KUKA KRL program: EPS_2_25862_MH7A_A_20251016034305.src

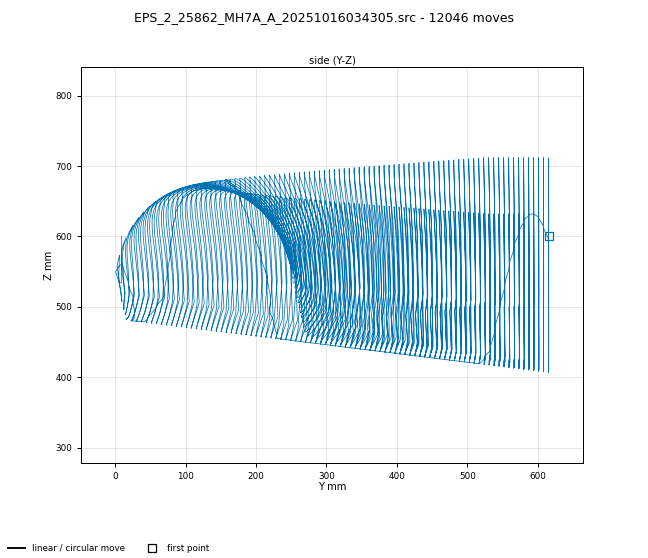
[picture p0: tool path of EPS_2_25862_MH7A_A_20251016034305.src, 12046 of 12048 moves have a stored position in this frame; points joined in program order, loops and branches not executed]
&ACCESS RVP
&REL 4
&COMMENT QRS 19112012
&PARAM EDITMASK = *
DEF PART()
EXT BAS (BAS_COMMAND :IN,REAL :IN )
INT I
BAS (#INITMOV,0 )

;KUKA QRS Post kuka4.cps  Date:22-06-2017 !

File_ID=2892

QRS_PRE_INIT()

;Init var - Until changes are made in qrs_pre_init
Outlet_Square_prg=0
Inlet_1_Square_prg=0
Inlet_2_Square_prg=0
Inlet_3_Square_prg=0
Inlet_4_Square_prg=0
Inlet_5_Square_prg=0

Outlet_1={X 0.000, Y 524.580, Z 611.500, B 0.000, E1 0.000 }
Inlet_1={X 0.000, Y 530.290, Z 531.500, B 0.000, E1 105.000 }
Outlet_1_type=201
Inlet_1_type=201
;QRS#1=Sidecore dimensions
;QRS#2=200-8" PVC SDR 35
;QRS#3=200-8" PVC SDR 35
;QRS#4=
;QRS#5=
;QRS#6=
;QRS#7=
;QRS#8=
;QRS#9=12-08 PSX
;QRS#10=12-08 PSX
;QRS#11=
;QRS#12=
;QRS#13=
;QRS#14=
;QRS#15=
;QRS#16=1220x127x991 3,25'
;QRS#17=EPS Height
;QRS#18=712
;QRS#19=*
;QRS#20= UPDATED VERSION 22-06-2017
;QRS#21=*
Outlet_Square=0100
Inlet_1_Square=0100
Inlet_2_Square=0
Inlet_3_Square=0
Inlet_4_Square=0
Inlet_5_Square=0
Mill_Square=1
Outlet_Square_Prg=204
Inlet_1_Square_prg=204

QRS_INIT()

$ADVANCE=5

; T1
PTP {E1 173.735,E2 173.735}
PTP {X 0,Y 615.512,A -85,B 0,C 180,E1 173.735,E2 173.735,E3 0,E4 0,E5 0,E6 0}
QRS_SPEED_INIT()
LIN {X 0,Y 615.512,Z 600,A -85,B 0,C 180,E1 173.735,E2 173.735,E3 0,E4 0,E5 0,E6 0} C_VEL
LIN {X 0,Y 615.512,Z 594.49,A -85,B 0,C 180,E1 173.735,E2 173.735} C_VEL
LIN {X 0,Y 615.498,Z 593.072,A -85,B 0,C 180,E1 173.417,E2 173.417} C_VEL
LIN {X 0,Y 615.497,Z 602.544,A -85,B 0,C 180,E1 172.455,E2 172.455} C_VEL
LIN {X 0,Y 615.496,Z 610.413,A -85,B 0,C 180,E1 171.464,E2 171.464} C_VEL
LIN {X 0,Y 615.497,Z 616.705,A -85,B 0,C 180,E1 170.47,E2 170.47} C_VEL
LIN {X 0,Y 615.496,Z 621.726,A -85,B 0,C 180,E1 169.473,E2 169.473} C_VEL
LIN {X 0,Y 615.496,Z 625.613,A -85,B 0,C 180,E1 168.473,E2 168.473} C_VEL
LIN {X 0,Y 615.495,Z 628.469,A -85,B 0,C 180,E1 167.47,E2 167.47} C_VEL
LIN {X 0,Y 615.496,Z 629.806,A -85,B 0,C 180,E1 166.799,E2 166.799} C_VEL
LIN {X 0,Y 615.497,Z 630.814,A -85,B 0,C 180,E1 166.065,E2 166.065} C_VEL
LIN {X 0,Y 615.494,Z 631.275,A -85,B 0,C 180,E1 165.451,E2 165.451} C_VEL
LIN {X 0,Y 615.496,Z 631.351,A -85,B 0,C 180,E1 164.774,E2 164.774} C_VEL
LIN {X 0,Y 615.495,Z 630.488,A -85,B 0,C 180,E1 163.568,E2 163.568} C_VEL
LIN {X 0,Y 615.495,Z 629.096,A -85,B 0,C 180,E1 162.73,E2 162.73} C_VEL
LIN {X 0,Y 615.497,Z 627.447,A -85,B 0,C 180,E1 162.043,E2 162.043} C_VEL
LIN {X 0,Y 615.496,Z 624.074,A -85,B 0,C 180,E1 161.009,E2 161.009} C_VEL
LIN {X 0,Y 615.496,Z 619.508,A -85,B 0,C 180,E1 159.968,E2 159.968} C_VEL
LIN {X 0,Y 615.496,Z 613.587,A -85,B 0,C 180,E1 158.919,E2 158.919} C_VEL
LIN {X 0,Y 615.498,Z 605.985,A -85,B 0,C 180,E1 157.864,E2 157.864} C_VEL
LIN {X 0,Y 615.498,Z 598.1,A -85,B 0,C 180,E1 156.978,E2 156.978} C_VEL
LIN {X 0,Y 615.497,Z 588.587,A -85,B 0,C 180,E1 156.104,E2 156.104} C_VEL
LIN {X 0,Y 615.479,Z 578.677,A -85,B 0,C 180,E1 155.368,E2 155.368} C_VEL
LIN {X 0,Y 615.462,Z 567.861,A -85,B 0,C 180,E1 154.72,E2 154.72} C_VEL
LIN {X 0,Y 615.492,Z 555.657,A -85,B 0,C 180,E1 154.148,E2 154.148} C_VEL
LIN {X 0,Y 615.484,Z 544.011,A -85,B 0,C 180,E1 153.738,E2 153.738} C_VEL
LIN {X 0,Y 615.481,Z 531.052,A -85,B 0,C 180,E1 153.424,E2 153.424} C_VEL
LIN {X 0,Y 615.492,Z 513.299,A -85,B 0,C 180,E1 153.181,E2 153.181} C_VEL
LIN {X 0,Y 615.484,Z 422.14,A -85,B 0,C 180,E1 152.108,E2 152.108} C_VEL
LIN {X 0,Y 615.478,Z 408.507,A -85,B 0,C 180,E1 149.46,E2 149.46} C_VEL
LIN {X 0,Y 615.445,Z 406.696,A -85,B 0,C 180,E1 149.078,E2 149.078} C_VEL
LIN {X 0,Y 615.439,Z 406.693,A -85,B 0,C 180,E1 146.761,E2 146.761} C_VEL
LIN {X 0,Y 615.478,Z 406.688,A -85,B 0,C 180,E1 144.168,E2 144.168} C_VEL
LIN {X 0,Y 615.489,Z 406.691,A -85,B 0,C 180,E1 141.932,E2 141.932} C_VEL
LIN {X 0,Y 615.473,Z 406.698,A -85,B 0,C 180,E1 139.392,E2 139.392} C_VEL
LIN {X 0,Y 615.443,Z 406.695,A -85,B 0,C 180,E1 136.958,E2 136.958} C_VEL
LIN {X 0,Y 615.442,Z 406.694,A -85,B 0,C 180,E1 134.927,E2 134.927} C_VEL
LIN {X 0,Y 615.485,Z 406.688,A -85,B 0,C 180,E1 132.08,E2 132.08} C_VEL
LIN {X 0,Y 615.493,Z 406.695,A -85,B 0,C 180,E1 129.75,E2 129.75} C_VEL
LIN {X 0,Y 615.444,Z 406.694,A -85,B 0,C 180,E1 126.931,E2 126.931} C_VEL
LIN {X 0,Y 615.443,Z 406.692,A -85,B 0,C 180,E1 124.694,E2 124.694} C_VEL
LIN {X 0,Y 615.46,Z 406.689,A -85,B 0,C 180,E1 122.326,E2 122.326} C_VEL
LIN {X 0,Y 615.479,Z 406.699,A -85,B 0,C 180,E1 119.407,E2 119.407} C_VEL
LIN {X 0,Y 615.447,Z 406.696,A -85,B 0,C 180,E1 117.037,E2 117.037} C_VEL
LIN {X 0,Y 615.448,Z 406.695,A -85,B 0,C 180,E1 114.994,E2 114.994} C_VEL
LIN {X 0,Y 615.462,Z 406.689,A -85,B 0,C 180,E1 112.34,E2 112.34} C_VEL
LIN {X 0,Y 615.474,Z 406.698,A -85,B 0,C 180,E1 109.339,E2 109.339} C_VEL
LIN {X 0,Y 615.468,Z 406.697,A -85,B 0,C 180,E1 107.271,E2 107.271} C_VEL
LIN {X 0,Y 615.464,Z 406.697,A -85,B 0,C 180,E1 105.227,E2 105.227} C_VEL
LIN {X 0,Y 615.462,Z 406.697,A -85,B 0,C 180,E1 103.202,E2 103.202} C_VEL
LIN {X 0,Y 615.446,Z 406.693,A -85,B 0,C 180,E1 100.867,E2 100.867} C_VEL
LIN {X 0,Y 615.45,Z 406.69,A -85,B 0,C 180,E1 98.537,E2 98.537} C_VEL
LIN {X 0,Y 615.495,Z 406.688,A -85,B 0,C 180,E1 95.899,E2 95.899} C_VEL
LIN {X 0,Y 615.471,Z 406.698,A -85,B 0,C 180,E1 93.273,E2 93.273} C_VEL
LIN {X 0,Y 615.448,Z 406.691,A -85,B 0,C 180,E1 90.655,E2 90.655} C_VEL
LIN {X 0,Y 615.495,Z 406.685,A -85,B 0,C 180,E1 88.037,E2 88.037} C_VEL
LIN {X 0,Y 615.489,Z 406.699,A -85,B 0,C 180,E1 85.416,E2 85.416} C_VEL
LIN {X 0,Y 615.446,Z 406.693,A -85,B 0,C 180,E1 82.784,E2 82.784} C_VEL
LIN {X 0,Y 615.481,Z 406.686,A -85,B 0,C 180,E1 80.138,E2 80.138} C_VEL
LIN {X 0,Y 615.487,Z 406.702,A -85,B 0,C 180,E1 77.47,E2 77.47} C_VEL
LIN {X 0,Y 615.446,Z 406.693,A -85,B 0,C 180,E1 74.773,E2 74.773} C_VEL
LIN {X 0,Y 615.49,Z 406.685,A -85,B 0,C 180,E1 72.043,E2 72.043} C_VEL
LIN {X 0,Y 615.474,Z 406.698,A -85,B 0,C 180,E1 69.269,E2 69.269} C_VEL
LIN {X 0,Y 615.466,Z 406.697,A -85,B 0,C 180,E1 67.155,E2 67.155} C_VEL
LIN {X 0,Y 615.457,Z 406.695,A -85,B 0,C 180,E1 65.007,E2 65.007} C_VEL
LIN {X 0,Y 615.451,Z 406.693,A -85,B 0,C 180,E1 62.821,E2 62.821} C_VEL
LIN {X 0,Y 615.476,Z 406.686,A -85,B 0,C 180,E1 60.208,E2 60.208} C_VEL
LIN {X 0,Y 615.493,Z 406.698,A -85,B 0,C 180,E1 57.543,E2 57.543} C_VEL
LIN {X 0,Y 615.471,Z 406.697,A -85,B 0,C 180,E1 55.184,E2 55.184} C_VEL
LIN {X 0,Y 615.451,Z 406.692,A -85,B 0,C 180,E1 52.755,E2 52.755} C_VEL
LIN {X 0,Y 615.496,Z 406.686,A -85,B 0,C 180,E1 49.91,E2 49.91} C_VEL
LIN {X 0,Y 615.493,Z 406.694,A -85,B 0,C 180,E1 47.648,E2 47.648} C_VEL
LIN {X 0,Y 615.457,Z 406.694,A -85,B 0,C 180,E1 44.929,E2 44.929} C_VEL
LIN {X 0,Y 615.487,Z 406.684,A -85,B 0,C 180,E1 42.08,E2 42.08} C_VEL
LIN {X 0,Y 615.489,Z 406.691,A -85,B 0,C 180,E1 39.75,E2 39.75} C_VEL
LIN {X 0,Y 615.458,Z 406.694,A -85,B 0,C 180,E1 36.933,E2 36.933} C_VEL
LIN {X 0,Y 615.454,Z 406.691,A -85,B 0,C 180,E1 34.696,E2 34.696} C_VEL
LIN {X 0,Y 615.465,Z 406.687,A -85,B 0,C 180,E1 32.328,E2 32.328} C_VEL
LIN {X 0,Y 615.49,Z 406.702,A -85,B 0,C 180,E1 29.406,E2 29.406} C_VEL
LIN {X 0,Y 615.464,Z 406.696,A -85,B 0,C 180,E1 27.041,E2 27.041} C_VEL
LIN {X 0,Y 615.463,Z 406.695,A -85,B 0,C 180,E1 24.993,E2 24.993} C_VEL
LIN {X 0,Y 615.466,Z 406.687,A -85,B 0,C 180,E1 22.341,E2 22.341} C_VEL
LIN {X 0,Y 615.484,Z 406.685,A -85,B 0,C 180,E1 20.033,E2 20.033} C_VEL
LIN {X 0,Y 615.487,Z 406.699,A -85,B 0,C 180,E1 17.271,E2 17.271} C_VEL
LIN {X 0,Y 615.456,Z 406.689,A -85,B 0,C 180,E1 14.55,E2 14.55} C_VEL
LIN {X 0,Y 615.494,Z 406.686,A -85,B 0,C 180,E1 11.861,E2 11.861} C_VEL
LIN {X 0,Y 615.482,Z 406.698,A -85,B 0,C 180,E1 9.199,E2 9.199} C_VEL
LIN {X 0,Y 615.458,Z 406.689,A -85,B 0,C 180,E1 6.555,E2 6.555} C_VEL
LIN {X 0,Y 615.489,Z 406.685,A -85,B 0,C 180,E1 3.928,E2 3.928} C_VEL
LIN {X 0,Y 615.494,Z 406.7,A -85,B 0,C 180,E1 1.309,E2 1.309} C_VEL
LIN {X 0,Y 615.458,Z 406.691,A -85,B 0,C 180,E1 -1.309,E2 -1.309} C_VEL
LIN {X 0,Y 615.485,Z 406.684,A -85,B 0,C 180,E1 -3.929,E2 -3.929} C_VEL
LIN {X 0,Y 615.489,Z 406.699,A -85,B 0,C 180,E1 -6.579,E2 -6.579} C_VEL
LIN {X 0,Y 615.46,Z 406.693,A -85,B 0,C 180,E1 -9.199,E2 -9.199} C_VEL
LIN {X 0,Y 615.485,Z 406.683,A -85,B 0,C 180,E1 -11.861,E2 -11.861} C_VEL
LIN {X 0,Y 615.489,Z 406.698,A -85,B 0,C 180,E1 -14.549,E2 -14.549} C_VEL
LIN {X 0,Y 615.458,Z 406.692,A -85,B 0,C 180,E1 -17.271,E2 -17.271} C_VEL
LIN {X 0,Y 615.489,Z 406.684,A -85,B 0,C 180,E1 -20.033,E2 -20.033} C_VEL
LIN {X 0,Y 615.484,Z 406.698,A -85,B 0,C 180,E1 -22.845,E2 -22.845} C_VEL
LIN {X 0,Y 615.465,Z 406.687,A -85,B 0,C 180,E1 -25.565,E2 -25.565} C_VEL
LIN {X 0,Y 615.484,Z 406.694,A -85,B 0,C 180,E1 -28.45,E2 -28.45} C_VEL
LIN {X 0,Y 615.468,Z 406.694,A -85,B 0,C 180,E1 -31.083,E2 -31.083} C_VEL
LIN {X 0,Y 615.464,Z 406.688,A -85,B 0,C 180,E1 -33.531,E2 -33.531} C_VEL
LIN {X 0,Y 615.483,Z 406.683,A -85,B 0,C 180,E1 -35.833,E2 -35.833} C_VEL
LIN {X 0,Y 615.487,Z 406.684,A -85,B 0,C 180,E1 -38.069,E2 -38.069} C_VEL
LIN {X 0,Y 615.485,Z 406.699,A -85,B 0,C 180,E1 -40.607,E2 -40.607} C_VEL
LIN {X 0,Y 615.464,Z 406.692,A -85,B 0,C 180,E1 -43.247,E2 -43.247} C_VEL
LIN {X 0,Y 615.487,Z 406.683,A -85,B 0,C 180,E1 -46.003,E2 -46.003} C_VEL
LIN {X 0,Y 615.48,Z 406.698,A -85,B 0,C 180,E1 -48.907,E2 -48.907} C_VEL
LIN {X 0,Y 615.471,Z 406.695,A -85,B 0,C 180,E1 -51.095,E2 -51.095} C_VEL
LIN {X 0,Y 615.467,Z 406.687,A -85,B 0,C 180,E1 -53.574,E2 -53.574} C_VEL
LIN {X 0,Y 615.487,Z 406.692,A -85,B 0,C 180,E1 -56.466,E2 -56.466} C_VEL
LIN {X 0,Y 615.47,Z 406.696,A -85,B 0,C 180,E1 -59.079,E2 -59.079} C_VEL
LIN {X 0,Y 615.467,Z 406.687,A -85,B 0,C 180,E1 -61.554,E2 -61.554} C_VEL
LIN {X 0,Y 615.486,Z 406.691,A -85,B 0,C 180,E1 -64.432,E2 -64.432} C_VEL
LIN {X 0,Y 615.49,Z 406.748,A -85,B 0,C 180,E1 -66.02,E2 -66.02} C_VEL
LIN {X 0,Y 615.457,Z 428.81,A -85,B 0,C 180,E1 -68.743,E2 -68.743} C_VEL
LIN {X 0,Y 615.492,Z 450.661,A -85,B 0,C 180,E1 -71.395,E2 -71.395} C_VEL
LIN {X 0,Y 615.489,Z 474.676,A -85,B 0,C 180,E1 -74.265,E2 -74.265} C_VEL
LIN {X 0,Y 615.443,Z 497.572,A -85,B 0,C 180,E1 -76.966,E2 -76.966} C_VEL
LIN {X 0,Y 615.447,Z 498.822,A -85,B 0,C 180,E1 -77.113,E2 -77.113} C_VEL
LIN {X 0,Y 615.467,Z 607.846,A -85,B 0,C 180,E1 -78.41,E2 -78.41} C_VEL
LIN {X 0,Y 615.463,Z 620.356,A -85,B 0,C 180,E1 -78.682,E2 -78.682} C_VEL
LIN {X 0,Y 615.484,Z 633.665,A -85,B 0,C 180,E1 -79.115,E2 -79.115} C_VEL
LIN {X 0,Y 615.486,Z 645.481,A -85,B 0,C 180,E1 -79.64,E2 -79.64} C_VEL
LIN {X 0,Y 615.492,Z 656.998,A -85,B 0,C 180,E1 -80.304,E2 -80.304} C_VEL
LIN {X 0,Y 615.499,Z 667.344,A -85,B 0,C 180,E1 -81.05,E2 -81.05} C_VEL
LIN {X 0,Y 615.498,Z 675.814,A -85,B 0,C 180,E1 -81.794,E2 -81.794} C_VEL
LIN {X 0,Y 615.498,Z 683.608,A -85,B 0,C 180,E1 -82.62,E2 -82.62} C_VEL
LIN {X 0,Y 615.496,Z 691.204,A -85,B 0,C 180,E1 -83.608,E2 -83.608} C_VEL
LIN {X 0,Y 615.498,Z 698.206,A -85,B 0,C 180,E1 -84.759,E2 -84.759} C_VEL
LIN {X 0,Y 615.494,Z 702.852,A -85,B 0,C 180,E1 -85.744,E2 -85.744} C_VEL
LIN {X 0,Y 615.494,Z 706.399,A -85,B 0,C 180,E1 -86.727,E2 -86.727} C_VEL
LIN {X 0,Y 615.497,Z 708.233,A -85,B 0,C 180,E1 -87.382,E2 -87.382} C_VEL
LIN {X 0,Y 615.499,Z 709.608,A -85,B 0,C 180,E1 -88.037,E2 -88.037} C_VEL
LIN {X 0,Y 615.496,Z 711.174,A -85,B 0,C 180,E1 -89.346,E2 -89.346} C_VEL
LIN {X 0,Y 615.494,Z 711.389,A -85,B 0,C 180,E1 -90,E2 -90} C_VEL
LIN {X 0,Y 615.495,Z 710.58,A -85,B 0,C 180,E1 -91.309,E2 -91.309} C_VEL
LIN {X 0,Y 615.499,Z 709.607,A -85,B 0,C 180,E1 -91.963,E2 -91.963} C_VEL
LIN {X 0,Y 615.497,Z 708.232,A -85,B 0,C 180,E1 -92.618,E2 -92.618} C_VEL
LIN {X 0,Y 615.496,Z 705.349,A -85,B 0,C 180,E1 -93.601,E2 -93.601} C_VEL
LIN {X 0,Y 615.498,Z 701.44,A -85,B 0,C 180,E1 -94.585,E2 -94.585} C_VEL
LIN {X 0,Y 615.499,Z 696.403,A -85,B 0,C 180,E1 -95.57,E2 -95.57} C_VEL
LIN {X 0,Y 615.497,Z 689.87,A -85,B 0,C 180,E1 -96.583,E2 -96.583} C_VEL
LIN {X 0,Y 615.497,Z 682.131,A -85,B 0,C 180,E1 -97.546,E2 -97.546} C_VEL
LIN {X 0,Y 615.498,Z 674.042,A -85,B 0,C 180,E1 -98.371,E2 -98.371} C_VEL
LIN {X 0,Y 615.499,Z 664.164,A -85,B 0,C 180,E1 -99.199,E2 -99.199} C_VEL
LIN {X 0,Y 615.491,Z 652.976,A -85,B 0,C 180,E1 -99.945,E2 -99.945} C_VEL
LIN {X 0,Y 615.487,Z 642.017,A -85,B 0,C 180,E1 -100.527,E2 -100.527} C_VEL
LIN {X 0,Y 615.473,Z 629.513,A -85,B 0,C 180,E1 -101.04,E2 -101.04} C_VEL
LIN {X 0,Y 615.463,Z 617.058,A -85,B 0,C 180,E1 -101.402,E2 -101.402} C_VEL
LIN {X 0,Y 615.47,Z 603.45,A -85,B 0,C 180,E1 -101.653,E2 -101.653} C_VEL
LIN {X 0,Y 615.447,Z 498.818,A -85,B 0,C 180,E1 -102.888,E2 -102.888} C_VEL
LIN {X 0,Y 615.492,Z 476.104,A -85,B 0,C 180,E1 -105.566,E2 -105.566} C_VEL
LIN {X 0,Y 615.494,Z 452.01,A -85,B 0,C 180,E1 -108.443,E2 -108.443} C_VEL
LIN {X 0,Y 615.447,Z 430.241,A -85,B 0,C 180,E1 -111.083,E2 -111.083} C_VEL
LIN {X 0,Y 615.487,Z 408.335,A -85,B 0,C 180,E1 -113.783,E2 -113.783} C_VEL
LIN {X 0,Y 615.492,Z 406.682,A -85,B 0,C 180,E1 -114.009,E2 -114.009} C_VEL
LIN {X 0,Y 615.471,Z 406.688,A -85,B 0,C 180,E1 -116.445,E2 -116.445} C_VEL
LIN {X 0,Y 615.471,Z 406.693,A -85,B 0,C 180,E1 -118.659,E2 -118.659} C_VEL
LIN {X 0,Y 615.484,Z 406.702,A -85,B 0,C 180,E1 -121.085,E2 -121.085} C_VEL
LIN {X 0,Y 615.493,Z 406.681,A -85,B 0,C 180,E1 -124.022,E2 -124.022} C_VEL
LIN {X 0,Y 615.485,Z 406.703,A -85,B 0,C 180,E1 -126.936,E2 -126.936} C_VEL
LIN {X 0,Y 615.476,Z 406.686,A -85,B 0,C 180,E1 -129.751,E2 -129.751} C_VEL
LIN {X 0,Y 615.485,Z 406.69,A -85,B 0,C 180,E1 -132.354,E2 -132.354} C_VEL
LIN {X 0,Y 615.471,Z 406.695,A -85,B 0,C 180,E1 -135.071,E2 -135.071} C_VEL
LIN {X 0,Y 615.488,Z 406.684,A -85,B 0,C 180,E1 -137.92,E2 -137.92} C_VEL
LIN {X 0,Y 615.491,Z 406.69,A -85,B 0,C 180,E1 -140.25,E2 -140.25} C_VEL
LIN {X 0,Y 615.456,Z 406.695,A -85,B 0,C 180,E1 -143.068,E2 -143.068} C_VEL
LIN {X 0,Y 615.449,Z 406.692,A -85,B 0,C 180,E1 -145.305,E2 -145.305} C_VEL
LIN {X 0,Y 615.461,Z 406.69,A -85,B 0,C 180,E1 -147.674,E2 -147.674} C_VEL
LIN {X 0,Y 615.473,Z 406.699,A -85,B 0,C 180,E1 -150.593,E2 -150.593} C_VEL
LIN {X 0,Y 615.44,Z 406.696,A -85,B 0,C 180,E1 -152.965,E2 -152.965} C_VEL
LIN {X 0,Y 615.432,Z 406.697,A -85,B 0,C 180,E1 -155.006,E2 -155.006} C_VEL
LIN {X 0,Y 615.429,Z 406.696,A -85,B 0,C 180,E1 -157.153,E2 -157.153} C_VEL
LIN {X 0,Y 615.483,Z 406.697,A -85,B 0,C 180,E1 -159.967,E2 -159.967} C_VEL
LIN {X 0,Y 615.428,Z 406.699,A -85,B 0,C 180,E1 -162.728,E2 -162.728} C_VEL
LIN {X 0,Y 615.42,Z 406.7,A -85,B 0,C 180,E1 -164.772,E2 -164.772} C_VEL
LIN {X 0,Y 615.415,Z 406.7,A -85,B 0,C 180,E1 -166.797,E2 -166.797} C_VEL
LIN {X 0,Y 615.416,Z 406.7,A -85,B 0,C 180,E1 -169.149,E2 -169.149} C_VEL
LIN {X 0,Y 615.442,Z 406.699,A -85,B 0,C 180,E1 -171.463,E2 -171.463} C_VEL
LIN {X 0,Y 615.483,Z 406.695,A -85,B 0,C 180,E1 -174.101,E2 -174.101} C_VEL
LIN {X 0,Y 615.43,Z 406.696,A -85,B 0,C 180,E1 -176.727,E2 -176.727} C_VEL
LIN {X 0,Y 615.442,Z 406.697,A -85,B 0,C 180,E1 -179.182,E2 -179.182} C_VEL
LIN {X 0,Y 615.474,Z 419.232,A -85,B 0,C 180,E1 -181.636,E2 -181.636} C_VEL
LIN {X 0,Y 615.482,Z 422.09,A -85,B 0,C 180,E1 -182.188,E2 -182.188} C_VEL
LIN {X 0,Y 615.485,Z 527.922,A -85,B 0,C 180,E1 -183.457,E2 -183.457} C_VEL
LIN {X 0,Y 615.482,Z 540.23,A -85,B 0,C 180,E1 -183.724,E2 -183.724} C_VEL
LIN {X 0,Y 615.496,Z 552.949,A -85,B 0,C 180,E1 -184.133,E2 -184.133} C_VEL
LIN {X 0,Y 615.468,Z 565.139,A -85,B 0,C 180,E1 -184.667,E2 -184.667} C_VEL
LIN {X 0,Y 615.471,Z 576.613,A -85,B 0,C 180,E1 -185.323,E2 -185.323} C_VEL
LIN {X 0,Y 615.498,Z 586.934,A -85,B 0,C 180,E1 -186.063,E2 -186.063} C_VEL
LIN {X 0,Y 615.498,Z 593.072,A -85,B 0,C 180,E1 -186.583,E2 -186.583} C_VEL
LIN {X 0,Y 614.841,Z 597.363,A -85,B 0,C 180,E1 -186.973,E2 -186.973} C_VEL
LIN {X 0,Y 611.975,Z 603.961,A -85,B 0,C 180,E1 -187.622,E2 -187.622} C_VEL
LIN {X 0,Y 609.116,Z 609.736,A -85,B 0,C 180,E1 -188.318,E2 -188.318} C_VEL
LIN {X 0,Y 608.449,Z 612.931,A -85,B 0,C 180,E1 -188.774,E2 -188.774} C_VEL
LIN {X 0,Y 608.433,Z 618.129,A -85,B 0,C 180,E1 -189.642,E2 -189.642} C_VEL
LIN {X 0,Y 608.437,Z 622.99,A -85,B 0,C 180,E1 -190.65,E2 -190.65} C_VEL
LIN {X 0,Y 608.436,Z 626.725,A -85,B 0,C 180,E1 -191.662,E2 -191.662} C_VEL
LIN {X 0,Y 608.419,Z 629.431,A -85,B 0,C 180,E1 -192.678,E2 -192.678} C_VEL
LIN {X 0,Y 608.439,Z 630.696,A -85,B 0,C 180,E1 -193.357,E2 -193.357} C_VEL
LIN {X 0,Y 608.435,Z 631.54,A -85,B 0,C 180,E1 -194.038,E2 -194.038} C_VEL
LIN {X 0,Y 608.424,Z 631.93,A -85,B 0,C 180,E1 -194.722,E2 -194.722} C_VEL
LIN {X 0,Y 608.419,Z 631.921,A -85,B 0,C 180,E1 -195.407,E2 -195.407} C_VEL
LIN {X 0,Y 608.422,Z 631.014,A -85,B 0,C 180,E1 -196.513,E2 -196.513} C_VEL
LIN {X 0,Y 608.42,Z 629.289,A -85,B 0,C 180,E1 -197.478,E2 -197.478} C_VEL
LIN {X 0,Y 608.429,Z 625.843,A -85,B 0,C 180,E1 -198.703,E2 -198.703} C_VEL
LIN {X 0,Y 608.435,Z 620.813,A -85,B 0,C 180,E1 -199.923,E2 -199.923} C_VEL
LIN {X 0,Y 608.452,Z 615.05,A -85,B 0,C 180,E1 -200.982,E2 -200.982} C_VEL
LIN {X 0,Y 608.456,Z 607.715,A -85,B 0,C 180,E1 -202.049,E2 -202.049} C_VEL
LIN {X 0,Y 608.457,Z 600.081,A -85,B 0,C 180,E1 -202.944,E2 -202.944} C_VEL
LIN {X 0,Y 608.482,Z 590.643,A -85,B 0,C 180,E1 -203.844,E2 -203.844} C_VEL
LIN {X 0,Y 608.479,Z 580.109,A -85,B 0,C 180,E1 -204.661,E2 -204.661} C_VEL
LIN {X 0,Y 608.468,Z 568.498,A -85,B 0,C 180,E1 -205.373,E2 -205.373} C_VEL
LIN {X 0,Y 608.508,Z 556.778,A -85,B 0,C 180,E1 -205.935,E2 -205.935} C_VEL
LIN {X 0,Y 608.526,Z 543.817,A -85,B 0,C 180,E1 -206.401,E2 -206.401} C_VEL
LIN {X 0,Y 608.537,Z 530.376,A -85,B 0,C 180,E1 -206.724,E2 -206.724} C_VEL
LIN {X 0,Y 608.556,Z 509.869,A -85,B 0,C 180,E1 -206.997,E2 -206.997} C_VEL
LIN {X 0,Y 608.446,Z 422.357,A -85,B 0,C 180,E1 -208.044,E2 -208.044} C_VEL
LIN {X 0,Y 608.451,Z 408.589,A -85,B 0,C 180,E1 -210.738,E2 -210.738} C_VEL
LIN {X 0,Y 608.416,Z 407.694,A -85,B 0,C 180,E1 -210.933,E2 -210.933} C_VEL
LIN {X 0,Y 608.437,Z 407.692,A -85,B 0,C 180,E1 -212.881,E2 -212.881} C_VEL
LIN {X 0,Y 608.416,Z 407.692,A -85,B 0,C 180,E1 -215.28,E2 -215.28} C_VEL
LIN {X 0,Y 608.465,Z 407.694,A -85,B 0,C 180,E1 -218.239,E2 -218.239} C_VEL
LIN {X 0,Y 608.412,Z 407.693,A -85,B 0,C 180,E1 -221.18,E2 -221.18} C_VEL
LIN {X 0,Y 608.465,Z 407.688,A -85,B 0,C 180,E1 -223.87,E2 -223.87} C_VEL
LIN {X 0,Y 608.452,Z 407.693,A -85,B 0,C 180,E1 -226.693,E2 -226.693} C_VEL
LIN {X 0,Y 608.426,Z 407.694,A -85,B 0,C 180,E1 -228.821,E2 -228.821} C_VEL
LIN {X 0,Y 608.457,Z 407.688,A -85,B 0,C 180,E1 -231.761,E2 -231.761} C_VEL
LIN {X 0,Y 608.434,Z 407.695,A -85,B 0,C 180,E1 -234.721,E2 -234.721} C_VEL
LIN {X 0,Y 608.434,Z 407.69,A -85,B 0,C 180,E1 -237.119,E2 -237.119} C_VEL
LIN {X 0,Y 608.471,Z 407.689,A -85,B 0,C 180,E1 -240.028,E2 -240.028} C_VEL
LIN {X 0,Y 608.454,Z 407.691,A -85,B 0,C 180,E1 -242.798,E2 -242.798} C_VEL
LIN {X 0,Y 608.431,Z 407.69,A -85,B 0,C 180,E1 -245.428,E2 -245.428} C_VEL
LIN {X 0,Y 608.467,Z 407.694,A -85,B 0,C 180,E1 -248.308,E2 -248.308} C_VEL
LIN {X 0,Y 608.438,Z 407.69,A -85,B 0,C 180,E1 -251.13,E2 -251.13} C_VEL
LIN {X 0,Y 608.455,Z 407.689,A -85,B 0,C 180,E1 -253.906,E2 -253.906} C_VEL
LIN {X 0,Y 608.449,Z 407.695,A -85,B 0,C 180,E1 -256.643,E2 -256.643} C_VEL
LIN {X 0,Y 608.43,Z 407.69,A -85,B 0,C 180,E1 -259.349,E2 -259.349} C_VEL
LIN {X 0,Y 608.48,Z 407.687,A -85,B 0,C 180,E1 -262.033,E2 -262.033} C_VEL
LIN {X 0,Y 608.451,Z 407.694,A -85,B 0,C 180,E1 -264.698,E2 -264.698} C_VEL
LIN {X 0,Y 608.444,Z 407.688,A -85,B 0,C 180,E1 -267.352,E2 -267.352} C_VEL
LIN {X 0,Y 608.477,Z 407.687,A -85,B 0,C 180,E1 -270,E2 -270} C_VEL
LIN {X 0,Y 608.474,Z 407.693,A -85,B 0,C 180,E1 -272.648,E2 -272.648} C_VEL
LIN {X 0,Y 608.433,Z 407.69,A -85,B 0,C 180,E1 -275.302,E2 -275.302} C_VEL
LIN {X 0,Y 608.475,Z 407.687,A -85,B 0,C 180,E1 -277.967,E2 -277.967} C_VEL
LIN {X 0,Y 608.429,Z 407.694,A -85,B 0,C 180,E1 -280.935,E2 -280.935} C_VEL
LIN {X 0,Y 608.437,Z 407.689,A -85,B 0,C 180,E1 -283.357,E2 -283.357} C_VEL
LIN {X 0,Y 608.46,Z 407.69,A -85,B 0,C 180,E1 -286.094,E2 -286.094} C_VEL
LIN {X 0,Y 608.448,Z 407.692,A -85,B 0,C 180,E1 -288.87,E2 -288.87} C_VEL
LIN {X 0,Y 608.453,Z 407.687,A -85,B 0,C 180,E1 -291.692,E2 -291.692} C_VEL
LIN {X 0,Y 608.446,Z 407.698,A -85,B 0,C 180,E1 -294.571,E2 -294.571} C_VEL
LIN {X 0,Y 608.431,Z 407.691,A -85,B 0,C 180,E1 -297.198,E2 -297.198} C_VEL
LIN {X 0,Y 608.461,Z 407.686,A -85,B 0,C 180,E1 -299.78,E2 -299.78} C_VEL
LIN {X 0,Y 608.466,Z 407.696,A -85,B 0,C 180,E1 -302.523,E2 -302.523} C_VEL
LIN {X 0,Y 608.425,Z 407.691,A -85,B 0,C 180,E1 -305.279,E2 -305.279} C_VEL
LIN {X 0,Y 608.466,Z 407.691,A -85,B 0,C 180,E1 -308.24,E2 -308.24} C_VEL
LIN {X 0,Y 608.424,Z 407.692,A -85,B 0,C 180,E1 -311.179,E2 -311.179} C_VEL
LIN {X 0,Y 608.466,Z 407.686,A -85,B 0,C 180,E1 -313.87,E2 -313.87} C_VEL
LIN {X 0,Y 608.468,Z 407.694,A -85,B 0,C 180,E1 -316.691,E2 -316.691} C_VEL
LIN {X 0,Y 608.44,Z 407.695,A -85,B 0,C 180,E1 -318.822,E2 -318.822} C_VEL
LIN {X 0,Y 608.46,Z 407.686,A -85,B 0,C 180,E1 -321.76,E2 -321.76} C_VEL
LIN {X 0,Y 608.447,Z 407.689,A -85,B 0,C 180,E1 -323.954,E2 -323.954} C_VEL
LIN {X 0,Y 608.47,Z 407.691,A -85,B 0,C 180,E1 -326.33,E2 -326.33} C_VEL
LIN {X 0,Y 608.443,Z 407.697,A -85,B 0,C 180,E1 -328.733,E2 -328.733} C_VEL
LIN {X 0,Y 608.449,Z 407.688,A -85,B 0,C 180,E1 -331.384,E2 -331.384} C_VEL
LIN {X 0,Y 608.437,Z 407.69,A -85,B 0,C 180,E1 -333.964,E2 -333.964} C_VEL
LIN {X 0,Y 608.473,Z 407.688,A -85,B 0,C 180,E1 -336.155,E2 -336.155} C_VEL
LIN {X 0,Y 608.444,Z 407.692,A -85,B 0,C 180,E1 -339.018,E2 -339.018} C_VEL
LIN {X 0,Y 608.444,Z 407.689,A -85,B 0,C 180,E1 -341.828,E2 -341.828} C_VEL
LIN {X 0,Y 608.467,Z 407.696,A -85,B 0,C 180,E1 -344.594,E2 -344.594} C_VEL
LIN {X 0,Y 608.454,Z 407.688,A -85,B 0,C 180,E1 -347.323,E2 -347.323} C_VEL
LIN {X 0,Y 608.456,Z 407.688,A -85,B 0,C 180,E1 -350.023,E2 -350.023} C_VEL
LIN {X 0,Y 608.462,Z 407.696,A -85,B 0,C 180,E1 -352.701,E2 -352.701} C_VEL
LIN {X 0,Y 608.467,Z 407.695,A -85,B 0,C 180,E1 -354.698,E2 -354.698} C_VEL
LIN {X 0,Y 608.452,Z 407.688,A -85,B 0,C 180,E1 -357.352,E2 -357.352} C_VEL
LIN {X 0,Y 608.477,Z 407.685,A -85,B 0,C 180,E1 -360,E2 -360} C_VEL
LIN {X 0,Y 608.48,Z 407.695,A -85,B 0,C 180,E1 -362.648,E2 -362.648} C_VEL
LIN {X 0,Y 608.443,Z 407.69,A -85,B 0,C 180,E1 -365.302,E2 -365.302} C_VEL
LIN {X 0,Y 608.477,Z 407.685,A -85,B 0,C 180,E1 -367.967,E2 -367.967} C_VEL
LIN {X 0,Y 608.465,Z 407.691,A -85,B 0,C 180,E1 -370.954,E2 -370.954} C_VEL
LIN {X 0,Y 608.446,Z 407.689,A -85,B 0,C 180,E1 -373.357,E2 -373.357} C_VEL
LIN {X 0,Y 608.461,Z 407.688,A -85,B 0,C 180,E1 -376.094,E2 -376.094} C_VEL
LIN {X 0,Y 608.452,Z 407.695,A -85,B 0,C 180,E1 -378.87,E2 -378.87} C_VEL
LIN {X 0,Y 608.457,Z 407.686,A -85,B 0,C 180,E1 -381.692,E2 -381.692} C_VEL
LIN {X 0,Y 608.449,Z 407.696,A -85,B 0,C 180,E1 -384.571,E2 -384.571} C_VEL
LIN {X 0,Y 608.442,Z 407.691,A -85,B 0,C 180,E1 -387.201,E2 -387.201} C_VEL
LIN {X 0,Y 608.465,Z 407.686,A -85,B 0,C 180,E1 -389.971,E2 -389.971} C_VEL
LIN {X 0,Y 608.448,Z 407.696,A -85,B 0,C 180,E1 -392.88,E2 -392.88} C_VEL
LIN {X 0,Y 608.435,Z 407.691,A -85,B 0,C 180,E1 -395.278,E2 -395.278} C_VEL
LIN {X 0,Y 608.468,Z 407.688,A -85,B 0,C 180,E1 -398.24,E2 -398.24} C_VEL
LIN {X 0,Y 608.437,Z 407.692,A -85,B 0,C 180,E1 -401.178,E2 -401.178} C_VEL
LIN {X 0,Y 608.467,Z 407.685,A -85,B 0,C 180,E1 -403.87,E2 -403.87} C_VEL
LIN {X 0,Y 608.483,Z 407.694,A -85,B 0,C 180,E1 -406.69,E2 -406.69} C_VEL
LIN {X 0,Y 608.451,Z 407.697,A -85,B 0,C 180,E1 -408.823,E2 -408.823} C_VEL
LIN {X 0,Y 608.431,Z 407.691,A -85,B 0,C 180,E1 -411.409,E2 -411.409} C_VEL
LIN {X 0,Y 608.448,Z 407.688,A -85,B 0,C 180,E1 -413.955,E2 -413.955} C_VEL
LIN {X 0,Y 608.466,Z 407.689,A -85,B 0,C 180,E1 -416.33,E2 -416.33} C_VEL
LIN {X 0,Y 608.448,Z 407.698,A -85,B 0,C 180,E1 -418.733,E2 -418.733} C_VEL
LIN {X 0,Y 608.456,Z 407.688,A -85,B 0,C 180,E1 -421.383,E2 -421.383} C_VEL
LIN {X 0,Y 608.438,Z 407.69,A -85,B 0,C 180,E1 -423.964,E2 -423.964} C_VEL
LIN {X 0,Y 608.48,Z 407.711,A -85,B 0,C 180,E1 -425.848,E2 -425.848} C_VEL
LIN {X 0,Y 608.595,Z 424.505,A -85,B 0,C 180,E1 -427.957,E2 -427.957} C_VEL
LIN {X 0,Y 608.525,Z 447.466,A -85,B 0,C 180,E1 -430.783,E2 -430.783} C_VEL
LIN {X 0,Y 608.505,Z 468.571,A -85,B 0,C 180,E1 -433.34,E2 -433.34} C_VEL
LIN {X 0,Y 608.503,Z 491.694,A -85,B 0,C 180,E1 -436.103,E2 -436.103} C_VEL
LIN {X 0,Y 608.478,Z 499.265,A -85,B 0,C 180,E1 -436.973,E2 -436.973} C_VEL
LIN {X 0,Y 608.531,Z 607.958,A -85,B 0,C 180,E1 -438.277,E2 -438.277} C_VEL
LIN {X 0,Y 608.498,Z 621.224,A -85,B 0,C 180,E1 -438.571,E2 -438.571} C_VEL
LIN {X 0,Y 608.512,Z 633.649,A -85,B 0,C 180,E1 -438.983,E2 -438.983} C_VEL
LIN {X 0,Y 608.504,Z 645.639,A -85,B 0,C 180,E1 -439.519,E2 -439.519} C_VEL
LIN {X 0,Y 608.483,Z 657.2,A -85,B 0,C 180,E1 -440.191,E2 -440.191} C_VEL
LIN {X 0,Y 608.485,Z 667.596,A -85,B 0,C 180,E1 -440.946,E2 -440.946} C_VEL
LIN {X 0,Y 608.475,Z 676.114,A -85,B 0,C 180,E1 -441.699,E2 -441.699} C_VEL
LIN {X 0,Y 608.471,Z 683.962,A -85,B 0,C 180,E1 -442.534,E2 -442.534} C_VEL
LIN {X 0,Y 608.461,Z 691.287,A -85,B 0,C 180,E1 -443.485,E2 -443.485} C_VEL
LIN {X 0,Y 608.45,Z 696.867,A -85,B 0,C 180,E1 -444.366,E2 -444.366} C_VEL
LIN {X 0,Y 608.432,Z 701.951,A -85,B 0,C 180,E1 -445.362,E2 -445.362} C_VEL
LIN {X 0,Y 608.449,Z 705.897,A -85,B 0,C 180,E1 -446.358,E2 -446.358} C_VEL
LIN {X 0,Y 608.425,Z 708.81,A -85,B 0,C 180,E1 -447.352,E2 -447.352} C_VEL
LIN {X 0,Y 608.444,Z 710.202,A -85,B 0,C 180,E1 -448.014,E2 -448.014} C_VEL
LIN {X 0,Y 608.438,Z 711.784,A -85,B 0,C 180,E1 -449.338,E2 -449.338} C_VEL
LIN {X 0,Y 608.434,Z 712,A -85,B 0,C 180,E1 -450,E2 -450} C_VEL
LIN {X 0,Y 608.448,Z 711.183,A -85,B 0,C 180,E1 -451.324,E2 -451.324} C_VEL
LIN {X 0,Y 608.444,Z 710.201,A -85,B 0,C 180,E1 -451.986,E2 -451.986} C_VEL
LIN {X 0,Y 608.425,Z 708.808,A -85,B 0,C 180,E1 -452.649,E2 -452.649} C_VEL
LIN {X 0,Y 608.449,Z 705.895,A -85,B 0,C 180,E1 -453.643,E2 -453.643} C_VEL
LIN {X 0,Y 608.432,Z 701.949,A -85,B 0,C 180,E1 -454.638,E2 -454.638} C_VEL
LIN {X 0,Y 608.437,Z 695.875,A -85,B 0,C 180,E1 -455.801,E2 -455.801} C_VEL
LIN {X 0,Y 608.462,Z 689.233,A -85,B 0,C 180,E1 -456.8,E2 -456.8} C_VEL
LIN {X 0,Y 608.456,Z 680.987,A -85,B 0,C 180,E1 -457.8,E2 -457.8} C_VEL
LIN {X 0,Y 608.472,Z 672.533,A -85,B 0,C 180,E1 -458.636,E2 -458.636} C_VEL
LIN {X 0,Y 608.478,Z 662.087,A -85,B 0,C 180,E1 -459.474,E2 -459.474} C_VEL
LIN {X 0,Y 608.501,Z 651.751,A -85,B 0,C 180,E1 -460.145,E2 -460.145} C_VEL
LIN {X 0,Y 608.517,Z 640.598,A -85,B 0,C 180,E1 -460.725,E2 -460.725} C_VEL
LIN {X 0,Y 608.515,Z 628.894,A -85,B 0,C 180,E1 -461.192,E2 -461.192} C_VEL
LIN {X 0,Y 608.528,Z 616.254,A -85,B 0,C 180,E1 -461.555,E2 -461.555} C_VEL
LIN {X 0,Y 608.533,Z 603.581,A -85,B 0,C 180,E1 -461.787,E2 -461.787} C_VEL
LIN {X 0,Y 608.446,Z 498.943,A -85,B 0,C 180,E1 -463.038,E2 -463.038} C_VEL
LIN {X 0,Y 608.503,Z 476.162,A -85,B 0,C 180,E1 -465.749,E2 -465.749} C_VEL
LIN {X 0,Y 608.558,Z 453.372,A -85,B 0,C 180,E1 -468.497,E2 -468.497} C_VEL
LIN {X 0,Y 608.537,Z 431.676,A -85,B 0,C 180,E1 -471.156,E2 -471.156} C_VEL
LIN {X 0,Y 608.622,Z 410.151,A -85,B 0,C 180,E1 -473.839,E2 -473.839} C_VEL
LIN {X 0,Y 608.47,Z 407.688,A -85,B 0,C 180,E1 -474.168,E2 -474.168} C_VEL
LIN {X 0,Y 608.446,Z 407.693,A -85,B 0,C 180,E1 -476.775,E2 -476.775} C_VEL
LIN {X 0,Y 608.471,Z 407.686,A -85,B 0,C 180,E1 -479.78,E2 -479.78} C_VEL
LIN {X 0,Y 608.454,Z 407.69,A -85,B 0,C 180,E1 -482.521,E2 -482.521} C_VEL
LIN {X 0,Y 608.453,Z 407.698,A -85,B 0,C 180,E1 -484.906,E2 -484.906} C_VEL
LIN {X 0,Y 608.467,Z 407.686,A -85,B 0,C 180,E1 -487.747,E2 -487.747} C_VEL
LIN {X 0,Y 608.455,Z 407.69,A -85,B 0,C 180,E1 -490.329,E2 -490.329} C_VEL
LIN {X 0,Y 608.445,Z 407.696,A -85,B 0,C 180,E1 -492.961,E2 -492.961} C_VEL
LIN {X 0,Y 608.454,Z 407.687,A -85,B 0,C 180,E1 -495.737,E2 -495.737} C_VEL
LIN {X 0,Y 608.459,Z 407.697,A -85,B 0,C 180,E1 -498.659,E2 -498.659} C_VEL
LIN {X 0,Y 608.461,Z 407.687,A -85,B 0,C 180,E1 -501.761,E2 -501.761} C_VEL
LIN {X 0,Y 608.436,Z 407.696,A -85,B 0,C 180,E1 -504.722,E2 -504.722} C_VEL
LIN {X 0,Y 608.438,Z 407.691,A -85,B 0,C 180,E1 -507.119,E2 -507.119} C_VEL
LIN {X 0,Y 608.471,Z 407.69,A -85,B 0,C 180,E1 -510.029,E2 -510.029} C_VEL
LIN {X 0,Y 608.426,Z 407.694,A -85,B 0,C 180,E1 -512.803,E2 -512.803} C_VEL
LIN {X 0,Y 608.42,Z 407.695,A -85,B 0,C 180,E1 -514.697,E2 -514.697} C_VEL
LIN {X 0,Y 608.416,Z 407.693,A -85,B 0,C 180,E1 -516.875,E2 -516.875} C_VEL
LIN {X 0,Y 608.428,Z 407.691,A -85,B 0,C 180,E1 -519.332,E2 -519.332} C_VEL
LIN {X 0,Y 608.436,Z 407.695,A -85,B 0,C 180,E1 -521.828,E2 -521.828} C_VEL
LIN {X 0,Y 608.426,Z 407.693,A -85,B 0,C 180,E1 -524.593,E2 -524.593} C_VEL
LIN {X 0,Y 608.412,Z 407.694,A -85,B 0,C 180,E1 -526.642,E2 -526.642} C_VEL
LIN {X 0,Y 608.385,Z 407.696,A -85,B 0,C 180,E1 -529.087,E2 -529.087} C_VEL
LIN {X 0,Y 608.414,Z 407.695,A -85,B 0,C 180,E1 -531.363,E2 -531.363} C_VEL
LIN {X 0,Y 608.453,Z 407.695,A -85,B 0,C 180,E1 -534.033,E2 -534.033} C_VEL
LIN {X 0,Y 608.403,Z 407.694,A -85,B 0,C 180,E1 -536.689,E2 -536.689} C_VEL
LIN {X 0,Y 608.422,Z 407.694,A -85,B 0,C 180,E1 -539.173,E2 -539.173} C_VEL
LIN {X 0,Y 608.443,Z 420.348,A -85,B 0,C 180,E1 -541.655,E2 -541.655} C_VEL
LIN {X 0,Y 608.446,Z 422.367,A -85,B 0,C 180,E1 -542.048,E2 -542.048} C_VEL
LIN {X 0,Y 608.533,Z 528.482,A -85,B 0,C 180,E1 -543.331,E2 -543.331} C_VEL
LIN {X 0,Y 608.542,Z 541.347,A -85,B 0,C 180,E1 -543.621,E2 -543.621} C_VEL
LIN {X 0,Y 608.537,Z 554.388,A -85,B 0,C 180,E1 -544.056,E2 -544.056} C_VEL
LIN {X 0,Y 608.474,Z 565.459,A -85,B 0,C 180,E1 -544.554,E2 -544.554} C_VEL
LIN {X 0,Y 608.457,Z 576.937,A -85,B 0,C 180,E1 -545.219,E2 -545.219} C_VEL
LIN {X 0,Y 608.498,Z 587.278,A -85,B 0,C 180,E1 -545.967,E2 -545.967} C_VEL
LIN {X 0,Y 608.463,Z 596.693,A -85,B 0,C 180,E1 -546.799,E2 -546.799} C_VEL
LIN {X 0,Y 608.455,Z 605.778,A -85,B 0,C 180,E1 -547.8,E2 -547.8} C_VEL
LIN {X 0,Y 608.449,Z 612.931,A -85,B 0,C 180,E1 -548.774,E2 -548.774} C_VEL
LIN {X 0,Y 607.782,Z 615.966,A -85,B 0,C 180,E1 -549.248,E2 -549.248} C_VEL
LIN {X 0,Y 604.898,Z 620.355,A -85,B 0,C 180,E1 -550.044,E2 -550.044} C_VEL
LIN {X 0,Y 602.005,Z 624.121,A -85,B 0,C 180,E1 -550.877,E2 -550.877} C_VEL
LIN {X 0,Y 601.332,Z 626.018,A -85,B 0,C 180,E1 -551.406,E2 -551.406} C_VEL
LIN {X 0,Y 601.338,Z 628.229,A -85,B 0,C 180,E1 -552.144,E2 -552.144} C_VEL
LIN {X 0,Y 601.325,Z 629.813,A -85,B 0,C 180,E1 -552.83,E2 -552.83} C_VEL
LIN {X 0,Y 601.353,Z 631.568,A -85,B 0,C 180,E1 -554.064,E2 -554.064} C_VEL
LIN {X 0,Y 601.319,Z 631.972,A -85,B 0,C 180,E1 -554.9,E2 -554.9} C_VEL
LIN {X 0,Y 601.326,Z 631.858,A -85,B 0,C 180,E1 -555.594,E2 -555.594} C_VEL
LIN {X 0,Y 601.322,Z 630.94,A -85,B 0,C 180,E1 -556.587,E2 -556.587} C_VEL
LIN {X 0,Y 601.314,Z 628.884,A -85,B 0,C 180,E1 -557.691,E2 -557.691} C_VEL
LIN {X 0,Y 601.348,Z 625.663,A -85,B 0,C 180,E1 -558.798,E2 -558.798} C_VEL
LIN {X 0,Y 601.336,Z 621.621,A -85,B 0,C 180,E1 -559.812,E2 -559.812} C_VEL
LIN {X 0,Y 601.382,Z 615.68,A -85,B 0,C 180,E1 -560.947,E2 -560.947} C_VEL
LIN {X 0,Y 601.377,Z 608.969,A -85,B 0,C 180,E1 -561.961,E2 -561.961} C_VEL
LIN {X 0,Y 601.405,Z 601.62,A -85,B 0,C 180,E1 -562.865,E2 -562.865} C_VEL
LIN {X 0,Y 601.446,Z 592.622,A -85,B 0,C 180,E1 -563.775,E2 -563.775} C_VEL
LIN {X 0,Y 601.458,Z 582.107,A -85,B 0,C 180,E1 -564.629,E2 -564.629} C_VEL
LIN {X 0,Y 601.446,Z 571.279,A -85,B 0,C 180,E1 -565.339,E2 -565.339} C_VEL
LIN {X 0,Y 601.544,Z 559.517,A -85,B 0,C 180,E1 -565.944,E2 -565.944} C_VEL
LIN {X 0,Y 601.569,Z 546.444,A -85,B 0,C 180,E1 -566.449,E2 -566.449} C_VEL
LIN {X 0,Y 601.591,Z 533.518,A -85,B 0,C 180,E1 -566.799,E2 -566.799} C_VEL
LIN {X 0,Y 601.614,Z 520.564,A -85,B 0,C 180,E1 -567.009,E2 -567.009} C_VEL
LIN {X 0,Y 601.529,Z 423.337,A -85,B 0,C 180,E1 -568.176,E2 -568.176} C_VEL
LIN {X 0,Y 601.388,Z 422.349,A -85,B 0,C 180,E1 -568.201,E2 -568.201} C_VEL
LIN {X 0,Y 601.393,Z 408.996,A -85,B 0,C 180,E1 -570.846,E2 -570.846} C_VEL
LIN {X 0,Y 601.389,Z 408.57,A -85,B 0,C 180,E1 -570.944,E2 -570.944} C_VEL
LIN {X 0,Y 601.41,Z 408.564,A -85,B 0,C 180,E1 -573.315,E2 -573.315} C_VEL
LIN {X 0,Y 601.394,Z 408.575,A -85,B 0,C 180,E1 -576.259,E2 -576.259} C_VEL
LIN {X 0,Y 601.384,Z 408.568,A -85,B 0,C 180,E1 -579.129,E2 -579.129} C_VEL
LIN {X 0,Y 601.419,Z 408.565,A -85,B 0,C 180,E1 -581.766,E2 -581.766} C_VEL
LIN {X 0,Y 601.401,Z 408.574,A -85,B 0,C 180,E1 -584.532,E2 -584.532} C_VEL
LIN {X 0,Y 601.372,Z 408.569,A -85,B 0,C 180,E1 -587.414,E2 -587.414} C_VEL
LIN {X 0,Y 601.402,Z 408.569,A -85,B 0,C 180,E1 -590.004,E2 -590.004} C_VEL
LIN {X 0,Y 601.402,Z 408.573,A -85,B 0,C 180,E1 -592.622,E2 -592.622} C_VEL
LIN {X 0,Y 601.381,Z 408.569,A -85,B 0,C 180,E1 -595.065,E2 -595.065} C_VEL
LIN {X 0,Y 601.405,Z 408.565,A -85,B 0,C 180,E1 -597.482,E2 -597.482} C_VEL
LIN {X 0,Y 601.409,Z 408.566,A -85,B 0,C 180,E1 -599.855,E2 -599.855} C_VEL
LIN {X 0,Y 601.399,Z 408.573,A -85,B 0,C 180,E1 -602.641,E2 -602.641} C_VEL
LIN {X 0,Y 601.387,Z 408.568,A -85,B 0,C 180,E1 -605.12,E2 -605.12} C_VEL
LIN {X 0,Y 601.399,Z 408.57,A -85,B 0,C 180,E1 -608.04,E2 -608.04} C_VEL
LIN {X 0,Y 601.409,Z 408.568,A -85,B 0,C 180,E1 -610.9,E2 -610.9} C_VEL
LIN {X 0,Y 601.414,Z 408.565,A -85,B 0,C 180,E1 -613.712,E2 -613.712} C_VEL
LIN {X 0,Y 601.409,Z 408.575,A -85,B 0,C 180,E1 -616.484,E2 -616.484} C_VEL
LIN {X 0,Y 601.388,Z 408.568,A -85,B 0,C 180,E1 -619.223,E2 -619.223} C_VEL
LIN {X 0,Y 601.439,Z 408.563,A -85,B 0,C 180,E1 -621.939,E2 -621.939} C_VEL
LIN {X 0,Y 601.417,Z 408.571,A -85,B 0,C 180,E1 -624.636,E2 -624.636} C_VEL
LIN {X 0,Y 601.413,Z 408.564,A -85,B 0,C 180,E1 -627.321,E2 -627.321} C_VEL
LIN {X 0,Y 601.445,Z 408.563,A -85,B 0,C 180,E1 -630,E2 -630} C_VEL
LIN {X 0,Y 601.437,Z 408.568,A -85,B 0,C 180,E1 -632.679,E2 -632.679} C_VEL
LIN {X 0,Y 601.401,Z 408.566,A -85,B 0,C 180,E1 -635.364,E2 -635.364} C_VEL
LIN {X 0,Y 601.438,Z 408.564,A -85,B 0,C 180,E1 -638.061,E2 -638.061} C_VEL
LIN {X 0,Y 601.405,Z 408.568,A -85,B 0,C 180,E1 -641.001,E2 -641.001} C_VEL
LIN {X 0,Y 601.4,Z 408.566,A -85,B 0,C 180,E1 -643.516,E2 -643.516} C_VEL
LIN {X 0,Y 601.441,Z 408.567,A -85,B 0,C 180,E1 -646.287,E2 -646.287} C_VEL
LIN {X 0,Y 601.41,Z 408.566,A -85,B 0,C 180,E1 -649.099,E2 -649.099} C_VEL
LIN {X 0,Y 601.395,Z 408.567,A -85,B 0,C 180,E1 -651.24,E2 -651.24} C_VEL
LIN {X 0,Y 601.463,Z 408.562,A -85,B 0,C 180,E1 -654.14,E2 -654.14} C_VEL
LIN {X 0,Y 601.393,Z 408.568,A -85,B 0,C 180,E1 -657.114,E2 -657.114} C_VEL
LIN {X 0,Y 601.396,Z 408.566,A -85,B 0,C 180,E1 -659.394,E2 -659.394} C_VEL
LIN {X 0,Y 601.398,Z 408.566,A -85,B 0,C 180,E1 -661.727,E2 -661.727} C_VEL
LIN {X 0,Y 601.42,Z 408.567,A -85,B 0,C 180,E1 -664.119,E2 -664.119} C_VEL
LIN {X 0,Y 601.392,Z 408.577,A -85,B 0,C 180,E1 -666.584,E2 -666.584} C_VEL
LIN {X 0,Y 601.396,Z 408.568,A -85,B 0,C 180,E1 -669.128,E2 -669.128} C_VEL
LIN {X 0,Y 601.42,Z 408.563,A -85,B 0,C 180,E1 -671.765,E2 -671.765} C_VEL
LIN {X 0,Y 601.425,Z 408.573,A -85,B 0,C 180,E1 -674.535,E2 -674.535} C_VEL
LIN {X 0,Y 601.38,Z 408.569,A -85,B 0,C 180,E1 -677.327,E2 -677.327} C_VEL
LIN {X 0,Y 601.401,Z 408.567,A -85,B 0,C 180,E1 -680.004,E2 -680.004} C_VEL
LIN {X 0,Y 601.432,Z 408.572,A -85,B 0,C 180,E1 -682.618,E2 -682.618} C_VEL
LIN {X 0,Y 601.39,Z 408.57,A -85,B 0,C 180,E1 -685.066,E2 -685.066} C_VEL
LIN {X 0,Y 601.41,Z 408.564,A -85,B 0,C 180,E1 -687.483,E2 -687.483} C_VEL
LIN {X 0,Y 601.429,Z 408.563,A -85,B 0,C 180,E1 -689.851,E2 -689.851} C_VEL
LIN {X 0,Y 601.42,Z 408.569,A -85,B 0,C 180,E1 -692.887,E2 -692.887} C_VEL
LIN {X 0,Y 601.457,Z 408.559,A -85,B 0,C 180,E1 -695.86,E2 -695.86} C_VEL
LIN {X 0,Y 601.403,Z 408.573,A -85,B 0,C 180,E1 -698.761,E2 -698.761} C_VEL
LIN {X 0,Y 601.411,Z 408.564,A -85,B 0,C 180,E1 -701.608,E2 -701.608} C_VEL
LIN {X 0,Y 601.41,Z 408.571,A -85,B 0,C 180,E1 -704.409,E2 -704.409} C_VEL
LIN {X 0,Y 601.404,Z 408.567,A -85,B 0,C 180,E1 -707.171,E2 -707.171} C_VEL
LIN {X 0,Y 601.429,Z 408.563,A -85,B 0,C 180,E1 -709.905,E2 -709.905} C_VEL
LIN {X 0,Y 601.44,Z 408.571,A -85,B 0,C 180,E1 -712.615,E2 -712.615} C_VEL
LIN {X 0,Y 601.401,Z 408.567,A -85,B 0,C 180,E1 -715.308,E2 -715.308} C_VEL
LIN {X 0,Y 601.434,Z 408.563,A -85,B 0,C 180,E1 -717.991,E2 -717.991} C_VEL
LIN {X 0,Y 601.452,Z 408.57,A -85,B 0,C 180,E1 -720.67,E2 -720.67} C_VEL
LIN {X 0,Y 601.408,Z 408.566,A -85,B 0,C 180,E1 -723.35,E2 -723.35} C_VEL
LIN {X 0,Y 601.415,Z 408.565,A -85,B 0,C 180,E1 -726.037,E2 -726.037} C_VEL
LIN {X 0,Y 601.415,Z 408.574,A -85,B 0,C 180,E1 -728.738,E2 -728.738} C_VEL
LIN {X 0,Y 601.409,Z 408.565,A -85,B 0,C 180,E1 -731.459,E2 -731.459} C_VEL
LIN {X 0,Y 601.42,Z 408.566,A -85,B 0,C 180,E1 -734.206,E2 -734.206} C_VEL
LIN {X 0,Y 601.428,Z 408.568,A -85,B 0,C 180,E1 -736.986,E2 -736.986} C_VEL
LIN {X 0,Y 601.399,Z 408.566,A -85,B 0,C 180,E1 -739.81,E2 -739.81} C_VEL
LIN {X 0,Y 601.416,Z 408.573,A -85,B 0,C 180,E1 -742.606,E2 -742.606} C_VEL
LIN {X 0,Y 601.394,Z 408.574,A -85,B 0,C 180,E1 -744.879,E2 -744.879} C_VEL
LIN {X 0,Y 601.393,Z 408.568,A -85,B 0,C 180,E1 -747.358,E2 -747.358} C_VEL
LIN {X 0,Y 601.413,Z 408.565,A -85,B 0,C 180,E1 -749.394,E2 -749.394} C_VEL
LIN {X 0,Y 601.399,Z 408.566,A -85,B 0,C 180,E1 -751.727,E2 -751.727} C_VEL
LIN {X 0,Y 601.423,Z 408.565,A -85,B 0,C 180,E1 -754.119,E2 -754.119} C_VEL
LIN {X 0,Y 601.403,Z 408.574,A -85,B 0,C 180,E1 -756.583,E2 -756.583} C_VEL
LIN {X 0,Y 601.404,Z 408.569,A -85,B 0,C 180,E1 -759.127,E2 -759.127} C_VEL
LIN {X 0,Y 601.422,Z 408.563,A -85,B 0,C 180,E1 -761.766,E2 -761.766} C_VEL
LIN {X 0,Y 601.426,Z 408.57,A -85,B 0,C 180,E1 -764.535,E2 -764.535} C_VEL
LIN {X 0,Y 601.406,Z 408.567,A -85,B 0,C 180,E1 -767.329,E2 -767.329} C_VEL
LIN {X 0,Y 601.412,Z 408.565,A -85,B 0,C 180,E1 -770.005,E2 -770.005} C_VEL
LIN {X 0,Y 601.436,Z 408.57,A -85,B 0,C 180,E1 -772.618,E2 -772.618} C_VEL
LIN {X 0,Y 601.399,Z 408.571,A -85,B 0,C 180,E1 -775.067,E2 -775.067} C_VEL
LIN {X 0,Y 601.416,Z 408.564,A -85,B 0,C 180,E1 -777.484,E2 -777.484} C_VEL
LIN {X 0,Y 601.43,Z 408.562,A -85,B 0,C 180,E1 -779.852,E2 -779.852} C_VEL
LIN {X 0,Y 601.449,Z 408.569,A -85,B 0,C 180,E1 -782.889,E2 -782.889} C_VEL
LIN {X 0,Y 601.44,Z 408.581,A -85,B 0,C 180,E1 -785.658,E2 -785.658} C_VEL
LIN {X 0,Y 601.76,Z 411.59,A -85,B 0,C 180,E1 -786.056,E2 -786.056} C_VEL
LIN {X 0,Y 601.649,Z 431.68,A -85,B 0,C 180,E1 -788.59,E2 -788.59} C_VEL
LIN {X 0,Y 601.609,Z 453.123,A -85,B 0,C 180,E1 -791.251,E2 -791.251} C_VEL
LIN {X 0,Y 601.532,Z 477.601,A -85,B 0,C 180,E1 -794.238,E2 -794.238} C_VEL
LIN {X 0,Y 601.436,Z 498.947,A -85,B 0,C 180,E1 -796.807,E2 -796.807} C_VEL
LIN {X 0,Y 601.634,Z 525.202,A -85,B 0,C 180,E1 -797.134,E2 -797.134} C_VEL
LIN {X 0,Y 601.602,Z 607.958,A -85,B 0,C 180,E1 -798.14,E2 -798.14} C_VEL
LIN {X 0,Y 601.562,Z 621.224,A -85,B 0,C 180,E1 -798.438,E2 -798.438} C_VEL
LIN {X 0,Y 601.543,Z 632.916,A -85,B 0,C 180,E1 -798.826,E2 -798.826} C_VEL
LIN {X 0,Y 601.516,Z 645.638,A -85,B 0,C 180,E1 -799.396,E2 -799.396} C_VEL
LIN {X 0,Y 601.484,Z 657.202,A -85,B 0,C 180,E1 -800.076,E2 -800.076} C_VEL
LIN {X 0,Y 601.444,Z 667.598,A -85,B 0,C 180,E1 -800.839,E2 -800.839} C_VEL
LIN {X 0,Y 601.429,Z 676.114,A -85,B 0,C 180,E1 -801.601,E2 -801.601} C_VEL
LIN {X 0,Y 601.418,Z 683.962,A -85,B 0,C 180,E1 -802.446,E2 -802.446} C_VEL
LIN {X 0,Y 601.37,Z 691.226,A -85,B 0,C 180,E1 -803.398,E2 -803.398} C_VEL
LIN {X 0,Y 601.372,Z 696.867,A -85,B 0,C 180,E1 -804.299,E2 -804.299} C_VEL
LIN {X 0,Y 601.336,Z 701.951,A -85,B 0,C 180,E1 -805.308,E2 -805.308} C_VEL
LIN {X 0,Y 601.368,Z 705.897,A -85,B 0,C 180,E1 -806.315,E2 -806.315} C_VEL
LIN {X 0,Y 601.325,Z 708.81,A -85,B 0,C 180,E1 -807.321,E2 -807.321} C_VEL
LIN {X 0,Y 601.343,Z 710.202,A -85,B 0,C 180,E1 -807.991,E2 -807.991} C_VEL
LIN {X 0,Y 601.339,Z 711.784,A -85,B 0,C 180,E1 -809.331,E2 -809.331} C_VEL
LIN {X 0,Y 601.335,Z 712,A -85,B 0,C 180,E1 -810,E2 -810} C_VEL
LIN {X 0,Y 601.347,Z 711.184,A -85,B 0,C 180,E1 -811.34,E2 -811.34} C_VEL
LIN {X 0,Y 601.343,Z 710.201,A -85,B 0,C 180,E1 -812.01,E2 -812.01} C_VEL
LIN {X 0,Y 601.325,Z 708.809,A -85,B 0,C 180,E1 -812.68,E2 -812.68} C_VEL
LIN {X 0,Y 601.368,Z 705.895,A -85,B 0,C 180,E1 -813.686,E2 -813.686} C_VEL
LIN {X 0,Y 601.336,Z 701.949,A -85,B 0,C 180,E1 -814.693,E2 -814.693} C_VEL
LIN {X 0,Y 601.372,Z 695.875,A -85,B 0,C 180,E1 -815.869,E2 -815.869} C_VEL
LIN {X 0,Y 601.382,Z 689.233,A -85,B 0,C 180,E1 -816.88,E2 -816.88} C_VEL
LIN {X 0,Y 601.401,Z 680.987,A -85,B 0,C 180,E1 -817.893,E2 -817.893} C_VEL
LIN {X 0,Y 601.436,Z 672.534,A -85,B 0,C 180,E1 -818.738,E2 -818.738} C_VEL
LIN {X 0,Y 601.448,Z 662.088,A -85,B 0,C 180,E1 -819.585,E2 -819.585} C_VEL
LIN {X 0,Y 601.478,Z 651.752,A -85,B 0,C 180,E1 -820.265,E2 -820.265} C_VEL
LIN {X 0,Y 601.535,Z 640.908,A -85,B 0,C 180,E1 -820.835,E2 -820.835} C_VEL
LIN {X 0,Y 601.545,Z 628.375,A -85,B 0,C 180,E1 -821.341,E2 -821.341} C_VEL
LIN {X 0,Y 601.554,Z 615.34,A -85,B 0,C 180,E1 -821.712,E2 -821.712} C_VEL
LIN {X 0,Y 601.61,Z 602.062,A -85,B 0,C 180,E1 -821.946,E2 -821.946} C_VEL
LIN {X 0,Y 601.466,Z 499.224,A -85,B 0,C 180,E1 -823.182,E2 -823.182} C_VEL
LIN {X 0,Y 601.532,Z 477.597,A -85,B 0,C 180,E1 -825.762,E2 -825.762} C_VEL
LIN {X 0,Y 601.61,Z 453.121,A -85,B 0,C 180,E1 -828.749,E2 -828.749} C_VEL
LIN {X 0,Y 601.65,Z 431.676,A -85,B 0,C 180,E1 -831.41,E2 -831.41} C_VEL
LIN {X 0,Y 601.76,Z 411.586,A -85,B 0,C 180,E1 -833.945,E2 -833.945} C_VEL
LIN {X 0,Y 601.422,Z 408.568,A -85,B 0,C 180,E1 -834.362,E2 -834.362} C_VEL
LIN {X 0,Y 601.454,Z 408.57,A -85,B 0,C 180,E1 -837.111,E2 -837.111} C_VEL
LIN {X 0,Y 601.432,Z 408.563,A -85,B 0,C 180,E1 -840.164,E2 -840.164} C_VEL
LIN {X 0,Y 601.417,Z 408.57,A -85,B 0,C 180,E1 -842.714,E2 -842.714} C_VEL
LIN {X 0,Y 601.397,Z 408.574,A -85,B 0,C 180,E1 -845.112,E2 -845.112} C_VEL
LIN {X 0,Y 601.437,Z 408.564,A -85,B 0,C 180,E1 -847.419,E2 -847.419} C_VEL
LIN {X 0,Y 601.404,Z 408.566,A -85,B 0,C 180,E1 -849.996,E2 -849.996} C_VEL
LIN {X 0,Y 601.411,Z 408.573,A -85,B 0,C 180,E1 -852.671,E2 -852.671} C_VEL
LIN {X 0,Y 601.402,Z 408.566,A -85,B 0,C 180,E1 -855.48,E2 -855.48} C_VEL
LIN {X 0,Y 601.425,Z 408.569,A -85,B 0,C 180,E1 -858.407,E2 -858.407} C_VEL
LIN {X 0,Y 601.4,Z 408.572,A -85,B 0,C 180,E1 -860.872,E2 -860.872} C_VEL
LIN {X 0,Y 601.389,Z 408.568,A -85,B 0,C 180,E1 -863.416,E2 -863.416} C_VEL
LIN {X 0,Y 601.435,Z 408.565,A -85,B 0,C 180,E1 -866.065,E2 -866.065} C_VEL
LIN {X 0,Y 601.395,Z 408.568,A -85,B 0,C 180,E1 -869.056,E2 -869.056} C_VEL
LIN {X 0,Y 601.399,Z 408.566,A -85,B 0,C 180,E1 -871.371,E2 -871.371} C_VEL
LIN {X 0,Y 601.414,Z 408.573,A -85,B 0,C 180,E1 -874.382,E2 -874.382} C_VEL
LIN {X 0,Y 601.38,Z 408.573,A -85,B 0,C 180,E1 -876.588,E2 -876.588} C_VEL
LIN {X 0,Y 601.399,Z 408.567,A -85,B 0,C 180,E1 -879.477,E2 -879.477} C_VEL
LIN {X 0,Y 601.373,Z 408.577,A -85,B 0,C 180,E1 -882.311,E2 -882.311} C_VEL
LIN {X 0,Y 601.378,Z 408.574,A -85,B 0,C 180,E1 -884.408,E2 -884.408} C_VEL
LIN {X 0,Y 601.379,Z 408.572,A -85,B 0,C 180,E1 -886.483,E2 -886.483} C_VEL
LIN {X 0,Y 601.352,Z 408.573,A -85,B 0,C 180,E1 -889.223,E2 -889.223} C_VEL
LIN {X 0,Y 601.428,Z 408.573,A -85,B 0,C 180,E1 -891.939,E2 -891.939} C_VEL
LIN {X 0,Y 601.385,Z 408.569,A -85,B 0,C 180,E1 -894.635,E2 -894.635} C_VEL
LIN {X 0,Y 601.411,Z 408.569,A -85,B 0,C 180,E1 -897.321,E2 -897.321} C_VEL
LIN {X 0,Y 601.402,Z 408.589,A -85,B 0,C 180,E1 -899.163,E2 -899.163} C_VEL
LIN {X 0,Y 601.405,Z 422.318,A -85,B 0,C 180,E1 -901.883,E2 -901.883} C_VEL
LIN {X 0,Y 601.661,Z 425.704,A -85,B 0,C 180,E1 -901.945,E2 -901.945} C_VEL
LIN {X 0,Y 601.599,Z 527.771,A -85,B 0,C 180,E1 -903.181,E2 -903.181} C_VEL
LIN {X 0,Y 601.559,Z 540.897,A -85,B 0,C 180,E1 -903.475,E2 -903.475} C_VEL
LIN {X 0,Y 601.545,Z 553.511,A -85,B 0,C 180,E1 -903.894,E2 -903.894} C_VEL
LIN {X 0,Y 601.497,Z 565.614,A -85,B 0,C 180,E1 -904.44,E2 -904.44} C_VEL
LIN {X 0,Y 601.441,Z 577.064,A -85,B 0,C 180,E1 -905.112,E2 -905.112} C_VEL
LIN {X 0,Y 601.466,Z 587.381,A -85,B 0,C 180,E1 -905.868,E2 -905.868} C_VEL
LIN {X 0,Y 601.415,Z 596.779,A -85,B 0,C 180,E1 -906.711,E2 -906.711} C_VEL
LIN {X 0,Y 601.396,Z 605.85,A -85,B 0,C 180,E1 -907.723,E2 -907.723} C_VEL
LIN {X 0,Y 601.383,Z 613.242,A -85,B 0,C 180,E1 -908.747,E2 -908.747} C_VEL
LIN {X 0,Y 601.344,Z 619.083,A -85,B 0,C 180,E1 -909.757,E2 -909.757} C_VEL
LIN {X 0,Y 601.354,Z 624.497,A -85,B 0,C 180,E1 -910.975,E2 -910.975} C_VEL
LIN {X 0,Y 601.332,Z 626.018,A -85,B 0,C 180,E1 -911.406,E2 -911.406} C_VEL
LIN {X 0,Y 600.675,Z 627.735,A -85,B 0,C 180,E1 -911.941,E2 -911.941} C_VEL
LIN {X 0,Y 597.845,Z 629.872,A -85,B 0,C 180,E1 -912.825,E2 -912.825} C_VEL
LIN {X 0,Y 595.424,Z 631.015,A -85,B 0,C 180,E1 -913.547,E2 -913.547} C_VEL
LIN {X 0,Y 594.342,Z 631.607,A -85,B 0,C 180,E1 -914.108,E2 -914.108} C_VEL
LIN {X 0,Y 594.231,Z 631.738,A -85,B 0,C 180,E1 -914.298,E2 -914.298} C_VEL
LIN {X 0,Y 594.213,Z 631.997,A -85,B 0,C 180,E1 -915.082,E2 -915.082} C_VEL
LIN {X 0,Y 594.224,Z 631.742,A -85,B 0,C 180,E1 -915.785,E2 -915.785} C_VEL
LIN {X 0,Y 594.238,Z 630.851,A -85,B 0,C 180,E1 -916.667,E2 -916.667} C_VEL
LIN {X 0,Y 594.209,Z 628.417,A -85,B 0,C 180,E1 -917.91,E2 -917.91} C_VEL
LIN {X 0,Y 594.248,Z 625.498,A -85,B 0,C 180,E1 -918.89,E2 -918.89} C_VEL
LIN {X 0,Y 594.262,Z 620.73,A -85,B 0,C 180,E1 -920.058,E2 -920.058} C_VEL
LIN {X 0,Y 594.318,Z 615.025,A -85,B 0,C 180,E1 -921.128,E2 -921.128} C_VEL
LIN {X 0,Y 594.312,Z 607.552,A -85,B 0,C 180,E1 -922.235,E2 -922.235} C_VEL
LIN {X 0,Y 594.369,Z 599.904,A -85,B 0,C 180,E1 -923.151,E2 -923.151} C_VEL
LIN {X 0,Y 594.394,Z 589.406,A -85,B 0,C 180,E1 -924.165,E2 -924.165} C_VEL
LIN {X 0,Y 594.458,Z 579.812,A -85,B 0,C 180,E1 -924.909,E2 -924.909} C_VEL
LIN {X 0,Y 594.479,Z 569.484,A -85,B 0,C 180,E1 -925.563,E2 -925.563} C_VEL
LIN {X 0,Y 594.563,Z 557.226,A -85,B 0,C 180,E1 -926.174,E2 -926.174} C_VEL
LIN {X 0,Y 594.599,Z 544.818,A -85,B 0,C 180,E1 -926.639,E2 -926.639} C_VEL
LIN {X 0,Y 594.639,Z 531.905,A -85,B 0,C 180,E1 -926.972,E2 -926.972} C_VEL
LIN {X 0,Y 594.695,Z 514.94,A -85,B 0,C 180,E1 -927.219,E2 -927.219} C_VEL
LIN {X 0,Y 594.591,Z 423.965,A -85,B 0,C 180,E1 -928.324,E2 -928.324} C_VEL
LIN {X 0,Y 594.351,Z 422.313,A -85,B 0,C 180,E1 -928.367,E2 -928.367} C_VEL
LIN {X 0,Y 594.338,Z 409.648,A -85,B 0,C 180,E1 -930.907,E2 -930.907} C_VEL
LIN {X 0,Y 594.378,Z 409.443,A -85,B 0,C 180,E1 -932.95,E2 -932.95} C_VEL
LIN {X 0,Y 594.321,Z 409.448,A -85,B 0,C 180,E1 -935.411,E2 -935.411} C_VEL
LIN {X 0,Y 594.373,Z 409.444,A -85,B 0,C 180,E1 -937.942,E2 -937.942} C_VEL
LIN {X 0,Y 594.361,Z 409.446,A -85,B 0,C 180,E1 -940.82,E2 -940.82} C_VEL
LIN {X 0,Y 594.351,Z 409.444,A -85,B 0,C 180,E1 -943.301,E2 -943.301} C_VEL
LIN {X 0,Y 594.347,Z 409.451,A -85,B 0,C 180,E1 -946.163,E2 -946.163} C_VEL
LIN {X 0,Y 594.373,Z 409.449,A -85,B 0,C 180,E1 -948.535,E2 -948.535} C_VEL
LIN {X 0,Y 594.366,Z 409.442,A -85,B 0,C 180,E1 -951.298,E2 -951.298} C_VEL
LIN {X 0,Y 594.347,Z 409.445,A -85,B 0,C 180,E1 -953.755,E2 -953.755} C_VEL
LIN {X 0,Y 594.377,Z 409.448,A -85,B 0,C 180,E1 -956.238,E2 -956.238} C_VEL
LIN {X 0,Y 594.364,Z 409.449,A -85,B 0,C 180,E1 -958.649,E2 -958.649} C_VEL
LIN {X 0,Y 594.375,Z 409.442,A -85,B 0,C 180,E1 -961.044,E2 -961.044} C_VEL
LIN {X 0,Y 594.369,Z 409.446,A -85,B 0,C 180,E1 -964.055,E2 -964.055} C_VEL
LIN {X 0,Y 594.364,Z 409.45,A -85,B 0,C 180,E1 -966.295,E2 -966.295} C_VEL
LIN {X 0,Y 594.383,Z 409.44,A -85,B 0,C 180,E1 -969.223,E2 -969.223} C_VEL
LIN {X 0,Y 594.339,Z 409.45,A -85,B 0,C 180,E1 -972.094,E2 -972.094} C_VEL
LIN {X 0,Y 594.354,Z 409.45,A -85,B 0,C 180,E1 -974.218,E2 -974.218} C_VEL
LIN {X 0,Y 594.376,Z 409.449,A -85,B 0,C 180,E1 -976.321,E2 -976.321} C_VEL
LIN {X 0,Y 594.353,Z 409.445,A -85,B 0,C 180,E1 -979.094,E2 -979.094} C_VEL
LIN {X 0,Y 594.381,Z 409.441,A -85,B 0,C 180,E1 -981.843,E2 -981.843} C_VEL
LIN {X 0,Y 594.383,Z 409.449,A -85,B 0,C 180,E1 -984.572,E2 -984.572} C_VEL
LIN {X 0,Y 594.382,Z 409.44,A -85,B 0,C 180,E1 -987.289,E2 -987.289} C_VEL
LIN {X 0,Y 594.414,Z 409.439,A -85,B 0,C 180,E1 -990,E2 -990} C_VEL
LIN {X 0,Y 594.4,Z 409.444,A -85,B 0,C 180,E1 -992.711,E2 -992.711} C_VEL
LIN {X 0,Y 594.369,Z 409.441,A -85,B 0,C 180,E1 -995.428,E2 -995.428} C_VEL
LIN {X 0,Y 594.383,Z 409.444,A -85,B 0,C 180,E1 -998.157,E2 -998.157} C_VEL
LIN {X 0,Y 594.375,Z 409.443,A -85,B 0,C 180,E1 -1001.065,E2 -1001.065} C_VEL
LIN {X 0,Y 594.371,Z 409.441,A -85,B 0,C 180,E1 -1003.679,E2 -1003.679} C_VEL
LIN {X 0,Y 594.376,Z 409.448,A -85,B 0,C 180,E1 -1006.713,E2 -1006.713} C_VEL
LIN {X 0,Y 594.361,Z 409.443,A -85,B 0,C 180,E1 -1009.334,E2 -1009.334} C_VEL
LIN {X 0,Y 594.358,Z 409.443,A -85,B 0,C 180,E1 -1011.503,E2 -1011.503} C_VEL
LIN {X 0,Y 594.39,Z 409.448,A -85,B 0,C 180,E1 -1014.446,E2 -1014.446} C_VEL
LIN {X 0,Y 594.356,Z 409.451,A -85,B 0,C 180,E1 -1016.701,E2 -1016.701} C_VEL
LIN {X 0,Y 594.376,Z 409.444,A -85,B 0,C 180,E1 -1018.999,E2 -1018.999} C_VEL
LIN {X 0,Y 594.373,Z 409.441,A -85,B 0,C 180,E1 -1021.642,E2 -1021.642} C_VEL
LIN {X 0,Y 594.371,Z 409.452,A -85,B 0,C 180,E1 -1024.58,E2 -1024.58} C_VEL
LIN {X 0,Y 594.386,Z 409.439,A -85,B 0,C 180,E1 -1027.608,E2 -1027.608} C_VEL
LIN {X 0,Y 594.369,Z 409.453,A -85,B 0,C 180,E1 -1030.567,E2 -1030.567} C_VEL
LIN {X 0,Y 594.35,Z 409.445,A -85,B 0,C 180,E1 -1033.301,E2 -1033.301} C_VEL
LIN {X 0,Y 594.36,Z 409.446,A -85,B 0,C 180,E1 -1036.161,E2 -1036.161} C_VEL
LIN {X 0,Y 594.379,Z 409.451,A -85,B 0,C 180,E1 -1038.536,E2 -1038.536} C_VEL
LIN {X 0,Y 594.368,Z 409.442,A -85,B 0,C 180,E1 -1041.297,E2 -1041.297} C_VEL
LIN {X 0,Y 594.347,Z 409.444,A -85,B 0,C 180,E1 -1043.755,E2 -1043.755} C_VEL
LIN {X 0,Y 594.379,Z 409.445,A -85,B 0,C 180,E1 -1046.239,E2 -1046.239} C_VEL
LIN {X 0,Y 594.367,Z 409.452,A -85,B 0,C 180,E1 -1048.65,E2 -1048.65} C_VEL
LIN {X 0,Y 594.375,Z 409.444,A -85,B 0,C 180,E1 -1051.044,E2 -1051.044} C_VEL
LIN {X 0,Y 594.366,Z 409.443,A -85,B 0,C 180,E1 -1053.3,E2 -1053.3} C_VEL
LIN {X 0,Y 594.388,Z 409.444,A -85,B 0,C 180,E1 -1056.296,E2 -1056.296} C_VEL
LIN {X 0,Y 594.388,Z 409.441,A -85,B 0,C 180,E1 -1059.224,E2 -1059.224} C_VEL
LIN {X 0,Y 594.352,Z 409.446,A -85,B 0,C 180,E1 -1062.095,E2 -1062.095} C_VEL
LIN {X 0,Y 594.359,Z 409.447,A -85,B 0,C 180,E1 -1064.219,E2 -1064.219} C_VEL
LIN {X 0,Y 594.382,Z 409.445,A -85,B 0,C 180,E1 -1066.321,E2 -1066.321} C_VEL
LIN {X 0,Y 594.359,Z 409.446,A -85,B 0,C 180,E1 -1069.094,E2 -1069.094} C_VEL
LIN {X 0,Y 594.411,Z 409.437,A -85,B 0,C 180,E1 -1071.843,E2 -1071.843} C_VEL
LIN {X 0,Y 594.398,Z 409.448,A -85,B 0,C 180,E1 -1074.572,E2 -1074.572} C_VEL
LIN {X 0,Y 594.39,Z 409.44,A -85,B 0,C 180,E1 -1077.289,E2 -1077.289} C_VEL
LIN {X 0,Y 594.414,Z 409.437,A -85,B 0,C 180,E1 -1080,E2 -1080} C_VEL
LIN {X 0,Y 594.409,Z 409.447,A -85,B 0,C 180,E1 -1082.711,E2 -1082.711} C_VEL
LIN {X 0,Y 594.377,Z 409.441,A -85,B 0,C 180,E1 -1085.428,E2 -1085.428} C_VEL
LIN {X 0,Y 594.414,Z 409.438,A -85,B 0,C 180,E1 -1088.157,E2 -1088.157} C_VEL
LIN {X 0,Y 594.39,Z 409.443,A -85,B 0,C 180,E1 -1091.074,E2 -1091.074} C_VEL
LIN {X 0,Y 594.375,Z 409.441,A -85,B 0,C 180,E1 -1093.679,E2 -1093.679} C_VEL
LIN {X 0,Y 594.396,Z 409.449,A -85,B 0,C 180,E1 -1096.72,E2 -1096.72} C_VEL
LIN {X 0,Y 594.364,Z 409.443,A -85,B 0,C 180,E1 -1099.335,E2 -1099.335} C_VEL
LIN {X 0,Y 594.362,Z 409.443,A -85,B 0,C 180,E1 -1101.504,E2 -1101.504} C_VEL
LIN {X 0,Y 594.39,Z 409.445,A -85,B 0,C 180,E1 -1104.446,E2 -1104.446} C_VEL
LIN {X 0,Y 594.369,Z 409.453,A -85,B 0,C 180,E1 -1106.7,E2 -1106.7} C_VEL
LIN {X 0,Y 594.381,Z 409.446,A -85,B 0,C 180,E1 -1108.999,E2 -1108.999} C_VEL
LIN {X 0,Y 594.375,Z 409.441,A -85,B 0,C 180,E1 -1111.642,E2 -1111.642} C_VEL
LIN {X 0,Y 594.38,Z 409.448,A -85,B 0,C 180,E1 -1114.58,E2 -1114.58} C_VEL
LIN {X 0,Y 594.388,Z 409.439,A -85,B 0,C 180,E1 -1117.608,E2 -1117.608} C_VEL
LIN {X 0,Y 594.37,Z 409.449,A -85,B 0,C 180,E1 -1120.567,E2 -1120.567} C_VEL
LIN {X 0,Y 594.365,Z 409.444,A -85,B 0,C 180,E1 -1123.3,E2 -1123.3} C_VEL
LIN {X 0,Y 594.376,Z 409.443,A -85,B 0,C 180,E1 -1126.16,E2 -1126.16} C_VEL
LIN {X 0,Y 594.375,Z 409.444,A -85,B 0,C 180,E1 -1129.179,E2 -1129.179} C_VEL
LIN {X 0,Y 594.383,Z 409.441,A -85,B 0,C 180,E1 -1132.059,E2 -1132.059} C_VEL
LIN {X 0,Y 594.35,Z 409.453,A -85,B 0,C 180,E1 -1134.677,E2 -1134.677} C_VEL
LIN {X 0,Y 594.377,Z 409.445,A -85,B 0,C 180,E1 -1137.089,E2 -1137.089} C_VEL
LIN {X 0,Y 594.387,Z 409.439,A -85,B 0,C 180,E1 -1139.672,E2 -1139.672} C_VEL
LIN {X 0,Y 594.377,Z 409.448,A -85,B 0,C 180,E1 -1142.539,E2 -1142.539} C_VEL
LIN {X 0,Y 594.379,Z 409.51,A -85,B 0,C 180,E1 -1145.47,E2 -1145.47} C_VEL
LIN {X 0,Y 594.899,Z 413.025,A -85,B 0,C 180,E1 -1145.948,E2 -1145.948} C_VEL
LIN {X 0,Y 594.74,Z 433.115,A -85,B 0,C 180,E1 -1148.511,E2 -1148.511} C_VEL
LIN {X 0,Y 594.671,Z 454.953,A -85,B 0,C 180,E1 -1151.252,E2 -1151.252} C_VEL
LIN {X 0,Y 594.56,Z 479.036,A -85,B 0,C 180,E1 -1154.225,E2 -1154.225} C_VEL
LIN {X 0,Y 594.465,Z 499.265,A -85,B 0,C 180,E1 -1156.661,E2 -1156.661} C_VEL
LIN {X 0,Y 594.725,Z 509.103,A -85,B 0,C 180,E1 -1156.786,E2 -1156.786} C_VEL
LIN {X 0,Y 594.654,Z 607.958,A -85,B 0,C 180,E1 -1157.999,E2 -1157.999} C_VEL
LIN {X 0,Y 594.626,Z 621.225,A -85,B 0,C 180,E1 -1158.301,E2 -1158.301} C_VEL
LIN {X 0,Y 594.588,Z 634.291,A -85,B 0,C 180,E1 -1158.746,E2 -1158.746} C_VEL
LIN {X 0,Y 594.532,Z 645.637,A -85,B 0,C 180,E1 -1159.27,E2 -1159.27} C_VEL
LIN {X 0,Y 594.472,Z 657.203,A -85,B 0,C 180,E1 -1159.958,E2 -1159.958} C_VEL
LIN {X 0,Y 594.414,Z 667.599,A -85,B 0,C 180,E1 -1160.73,E2 -1160.73} C_VEL
LIN {X 0,Y 594.383,Z 676.114,A -85,B 0,C 180,E1 -1161.501,E2 -1161.501} C_VEL
LIN {X 0,Y 594.347,Z 683.962,A -85,B 0,C 180,E1 -1162.356,E2 -1162.356} C_VEL
LIN {X 0,Y 594.282,Z 691.813,A -85,B 0,C 180,E1 -1163.408,E2 -1163.408} C_VEL
LIN {X 0,Y 594.289,Z 698.682,A -85,B 0,C 180,E1 -1164.572,E2 -1164.572} C_VEL
LIN {X 0,Y 594.27,Z 703.372,A -85,B 0,C 180,E1 -1165.592,E2 -1165.592} C_VEL
LIN {X 0,Y 594.267,Z 706.957,A -85,B 0,C 180,E1 -1166.61,E2 -1166.61} C_VEL
LIN {X 0,Y 594.226,Z 708.809,A -85,B 0,C 180,E1 -1167.289,E2 -1167.289} C_VEL
LIN {X 0,Y 594.241,Z 710.202,A -85,B 0,C 180,E1 -1167.967,E2 -1167.967} C_VEL
LIN {X 0,Y 594.239,Z 711.784,A -85,B 0,C 180,E1 -1169.323,E2 -1169.323} C_VEL
LIN {X 0,Y 594.236,Z 712,A -85,B 0,C 180,E1 -1170,E2 -1170} C_VEL
LIN {X 0,Y 594.247,Z 711.184,A -85,B 0,C 180,E1 -1171.356,E2 -1171.356} C_VEL
LIN {X 0,Y 594.241,Z 710.201,A -85,B 0,C 180,E1 -1172.034,E2 -1172.034} C_VEL
LIN {X 0,Y 594.226,Z 708.809,A -85,B 0,C 180,E1 -1172.712,E2 -1172.712} C_VEL
LIN {X 0,Y 594.289,Z 705.895,A -85,B 0,C 180,E1 -1173.73,E2 -1173.73} C_VEL
LIN {X 0,Y 594.241,Z 701.948,A -85,B 0,C 180,E1 -1174.749,E2 -1174.749} C_VEL
LIN {X 0,Y 594.304,Z 695.876,A -85,B 0,C 180,E1 -1175.94,E2 -1175.94} C_VEL
LIN {X 0,Y 594.308,Z 689.234,A -85,B 0,C 180,E1 -1176.962,E2 -1176.962} C_VEL
LIN {X 0,Y 594.36,Z 680.987,A -85,B 0,C 180,E1 -1177.987,E2 -1177.987} C_VEL
LIN {X 0,Y 594.382,Z 672.534,A -85,B 0,C 180,E1 -1178.842,E2 -1178.842} C_VEL
LIN {X 0,Y 594.431,Z 662.09,A -85,B 0,C 180,E1 -1179.7,E2 -1179.7} C_VEL
LIN {X 0,Y 594.489,Z 651.754,A -85,B 0,C 180,E1 -1180.387,E2 -1180.387} C_VEL
LIN {X 0,Y 594.559,Z 640.713,A -85,B 0,C 180,E1 -1180.974,E2 -1180.974} C_VEL
LIN {X 0,Y 594.573,Z 628.701,A -85,B 0,C 180,E1 -1181.465,E2 -1181.465} C_VEL
LIN {X 0,Y 594.608,Z 615.339,A -85,B 0,C 180,E1 -1181.851,E2 -1181.851} C_VEL
LIN {X 0,Y 594.675,Z 602.062,A -85,B 0,C 180,E1 -1182.088,E2 -1182.088} C_VEL
LIN {X 0,Y 594.565,Z 500.118,A -85,B 0,C 180,E1 -1183.327,E2 -1183.327} C_VEL
LIN {X 0,Y 594.432,Z 498.764,A -85,B 0,C 180,E1 -1183.373,E2 -1183.373} C_VEL
LIN {X 0,Y 594.568,Z 474.727,A -85,B 0,C 180,E1 -1186.304,E2 -1186.304} C_VEL
LIN {X 0,Y 594.667,Z 452.081,A -85,B 0,C 180,E1 -1189.106,E2 -1189.106} C_VEL
LIN {X 0,Y 594.829,Z 428.806,A -85,B 0,C 180,E1 -1192.033,E2 -1192.033} C_VEL
LIN {X 0,Y 594.853,Z 411.586,A -85,B 0,C 180,E1 -1194.24,E2 -1194.24} C_VEL
LIN {X 0,Y 594.37,Z 409.449,A -85,B 0,C 180,E1 -1194.573,E2 -1194.573} C_VEL
LIN {X 0,Y 594.379,Z 409.446,A -85,B 0,C 180,E1 -1197.461,E2 -1197.461} C_VEL
LIN {X 0,Y 594.39,Z 409.441,A -85,B 0,C 180,E1 -1200.328,E2 -1200.328} C_VEL
LIN {X 0,Y 594.379,Z 409.451,A -85,B 0,C 180,E1 -1202.951,E2 -1202.951} C_VEL
LIN {X 0,Y 594.353,Z 409.448,A -85,B 0,C 180,E1 -1205.409,E2 -1205.409} C_VEL
LIN {X 0,Y 594.389,Z 409.44,A -85,B 0,C 180,E1 -1207.941,E2 -1207.941} C_VEL
LIN {X 0,Y 594.377,Z 409.452,A -85,B 0,C 180,E1 -1210.822,E2 -1210.822} C_VEL
LIN {X 0,Y 594.355,Z 409.446,A -85,B 0,C 180,E1 -1213.301,E2 -1213.301} C_VEL
LIN {X 0,Y 594.365,Z 409.445,A -85,B 0,C 180,E1 -1216.161,E2 -1216.161} C_VEL
LIN {X 0,Y 594.372,Z 409.444,A -85,B 0,C 180,E1 -1219.179,E2 -1219.179} C_VEL
LIN {X 0,Y 594.382,Z 409.443,A -85,B 0,C 180,E1 -1222.059,E2 -1222.059} C_VEL
LIN {X 0,Y 594.33,Z 409.454,A -85,B 0,C 180,E1 -1224.68,E2 -1224.68} C_VEL
LIN {X 0,Y 594.376,Z 409.442,A -85,B 0,C 180,E1 -1227.09,E2 -1227.09} C_VEL
LIN {X 0,Y 594.372,Z 409.442,A -85,B 0,C 180,E1 -1229.675,E2 -1229.675} C_VEL
LIN {X 0,Y 594.346,Z 409.453,A -85,B 0,C 180,E1 -1232.482,E2 -1232.482} C_VEL
LIN {X 0,Y 594.335,Z 409.449,A -85,B 0,C 180,E1 -1234.805,E2 -1234.805} C_VEL
LIN {X 0,Y 594.352,Z 409.444,A -85,B 0,C 180,E1 -1237.269,E2 -1237.269} C_VEL
LIN {X 0,Y 594.351,Z 409.451,A -85,B 0,C 180,E1 -1239.945,E2 -1239.945} C_VEL
LIN {X 0,Y 594.321,Z 409.449,A -85,B 0,C 180,E1 -1242.804,E2 -1242.804} C_VEL
LIN {X 0,Y 594.37,Z 409.449,A -85,B 0,C 180,E1 -1245.836,E2 -1245.836} C_VEL
LIN {X 0,Y 594.353,Z 409.448,A -85,B 0,C 180,E1 -1248.403,E2 -1248.403} C_VEL
LIN {X 0,Y 594.325,Z 409.449,A -85,B 0,C 180,E1 -1251.157,E2 -1251.157} C_VEL
LIN {X 0,Y 594.352,Z 409.454,A -85,B 0,C 180,E1 -1253.891,E2 -1253.891} C_VEL
LIN {X 0,Y 594.314,Z 409.45,A -85,B 0,C 180,E1 -1256.61,E2 -1256.61} C_VEL
LIN {X 0,Y 594.381,Z 409.494,A -85,B 0,C 180,E1 -1259.153,E2 -1259.153} C_VEL
LIN {X 0,Y 594.342,Z 422.38,A -85,B 0,C 180,E1 -1261.736,E2 -1261.736} C_VEL
LIN {X 0,Y 594.747,Z 426.388,A -85,B 0,C 180,E1 -1261.799,E2 -1261.799} C_VEL
LIN {X 0,Y 594.644,Z 528.248,A -85,B 0,C 180,E1 -1263.049,E2 -1263.049} C_VEL
LIN {X 0,Y 594.613,Z 541.164,A -85,B 0,C 180,E1 -1263.346,E2 -1263.346} C_VEL
LIN {X 0,Y 594.569,Z 553.729,A -85,B 0,C 180,E1 -1263.77,E2 -1263.77} C_VEL
LIN {X 0,Y 594.5,Z 565.776,A -85,B 0,C 180,E1 -1264.322,E2 -1264.322} C_VEL
LIN {X 0,Y 594.426,Z 577.191,A -85,B 0,C 180,E1 -1265.002,E2 -1265.002} C_VEL
LIN {X 0,Y 594.434,Z 587.482,A -85,B 0,C 180,E1 -1265.768,E2 -1265.768} C_VEL
LIN {X 0,Y 594.379,Z 597.35,A -85,B 0,C 180,E1 -1266.67,E2 -1266.67} C_VEL
LIN {X 0,Y 594.324,Z 605.926,A -85,B 0,C 180,E1 -1267.645,E2 -1267.645} C_VEL
LIN {X 0,Y 594.313,Z 613.245,A -85,B 0,C 180,E1 -1268.672,E2 -1268.672} C_VEL
LIN {X 0,Y 594.272,Z 618.221,A -85,B 0,C 180,E1 -1269.53,E2 -1269.53} C_VEL
LIN {X 0,Y 594.289,Z 623.053,A -85,B 0,C 180,E1 -1270.562,E2 -1270.562} C_VEL
LIN {X 0,Y 594.246,Z 626.768,A -85,B 0,C 180,E1 -1271.599,E2 -1271.599} C_VEL
LIN {X 0,Y 594.237,Z 628.704,A -85,B 0,C 180,E1 -1272.291,E2 -1272.291} C_VEL
LIN {X 0,Y 594.244,Z 630.163,A -85,B 0,C 180,E1 -1272.986,E2 -1272.986} C_VEL
LIN {X 0,Y 594.231,Z 631.738,A -85,B 0,C 180,E1 -1274.298,E2 -1274.298} C_VEL
LIN {X 0,Y 593.5,Z 631.983,A -85,B 0,C 180,E1 -1274.863,E2 -1274.863} C_VEL
LIN {X 0,Y 590.615,Z 631.749,A -85,B 0,C 180,E1 -1275.78,E2 -1275.78} C_VEL
LIN {X 0,Y 588.222,Z 631.061,A -85,B 0,C 180,E1 -1276.516,E2 -1276.516} C_VEL
LIN {X 0,Y 587.207,Z 630.241,A -85,B 0,C 180,E1 -1277.081,E2 -1277.081} C_VEL
LIN {X 0,Y 587.129,Z 629.847,A -85,B 0,C 180,E1 -1277.271,E2 -1277.271} C_VEL
LIN {X 0,Y 587.161,Z 626.884,A -85,B 0,C 180,E1 -1278.493,E2 -1278.493} C_VEL
LIN {X 0,Y 587.155,Z 623.055,A -85,B 0,C 180,E1 -1279.582,E2 -1279.582} C_VEL
LIN {X 0,Y 587.186,Z 618.06,A -85,B 0,C 180,E1 -1280.657,E2 -1280.657} C_VEL
LIN {X 0,Y 587.23,Z 611.416,A -85,B 0,C 180,E1 -1281.778,E2 -1281.778} C_VEL
LIN {X 0,Y 587.262,Z 603.333,A -85,B 0,C 180,E1 -1282.854,E2 -1282.854} C_VEL
LIN {X 0,Y 587.324,Z 594.321,A -85,B 0,C 180,E1 -1283.82,E2 -1283.82} C_VEL
LIN {X 0,Y 587.392,Z 585.057,A -85,B 0,C 180,E1 -1284.633,E2 -1284.633} C_VEL
LIN {X 0,Y 587.433,Z 574.039,A -85,B 0,C 180,E1 -1285.417,E2 -1285.417} C_VEL
LIN {X 0,Y 587.556,Z 562.201,A -85,B 0,C 180,E1 -1286.077,E2 -1286.077} C_VEL
LIN {X 0,Y 587.622,Z 549.948,A -85,B 0,C 180,E1 -1286.6,E2 -1286.6} C_VEL
LIN {X 0,Y 587.682,Z 537.272,A -85,B 0,C 180,E1 -1286.993,E2 -1286.993} C_VEL
LIN {X 0,Y 587.729,Z 524.474,A -85,B 0,C 180,E1 -1287.243,E2 -1287.243} C_VEL
LIN {X 0,Y 587.69,Z 424.845,A -85,B 0,C 180,E1 -1288.472,E2 -1288.472} C_VEL
LIN {X 0,Y 587.31,Z 422.337,A -85,B 0,C 180,E1 -1288.525,E2 -1288.525} C_VEL
LIN {X 0,Y 587.319,Z 410.323,A -85,B 0,C 180,E1 -1290.967,E2 -1290.967} C_VEL
LIN {X 0,Y 587.329,Z 410.319,A -85,B 0,C 180,E1 -1293.397,E2 -1293.397} C_VEL
LIN {X 0,Y 587.281,Z 410.328,A -85,B 0,C 180,E1 -1295.901,E2 -1295.901} C_VEL
LIN {X 0,Y 587.317,Z 410.329,A -85,B 0,C 180,E1 -1298.48,E2 -1298.48} C_VEL
LIN {X 0,Y 587.31,Z 410.321,A -85,B 0,C 180,E1 -1301.159,E2 -1301.159} C_VEL
LIN {X 0,Y 587.301,Z 410.325,A -85,B 0,C 180,E1 -1303.953,E2 -1303.953} C_VEL
LIN {X 0,Y 587.288,Z 410.327,A -85,B 0,C 180,E1 -1306.885,E2 -1306.885} C_VEL
LIN {X 0,Y 587.306,Z 410.323,A -85,B 0,C 180,E1 -1309.744,E2 -1309.744} C_VEL
LIN {X 0,Y 587.321,Z 410.33,A -85,B 0,C 180,E1 -1312.39,E2 -1312.39} C_VEL
LIN {X 0,Y 587.338,Z 410.318,A -85,B 0,C 180,E1 -1315.654,E2 -1315.654} C_VEL
LIN {X 0,Y 587.334,Z 410.325,A -85,B 0,C 180,E1 -1318.23,E2 -1318.23} C_VEL
LIN {X 0,Y 587.344,Z 410.32,A -85,B 0,C 180,E1 -1320.868,E2 -1320.868} C_VEL
LIN {X 0,Y 587.31,Z 410.322,A -85,B 0,C 180,E1 -1323.829,E2 -1323.829} C_VEL
LIN {X 0,Y 587.305,Z 410.325,A -85,B 0,C 180,E1 -1325.992,E2 -1325.992} C_VEL
LIN {X 0,Y 587.334,Z 410.32,A -85,B 0,C 180,E1 -1328.962,E2 -1328.962} C_VEL
LIN {X 0,Y 587.289,Z 410.325,A -85,B 0,C 180,E1 -1331.872,E2 -1331.872} C_VEL
LIN {X 0,Y 587.303,Z 410.325,A -85,B 0,C 180,E1 -1334.024,E2 -1334.024} C_VEL
LIN {X 0,Y 587.356,Z 410.32,A -85,B 0,C 180,E1 -1336.154,E2 -1336.154} C_VEL
LIN {X 0,Y 587.34,Z 410.32,A -85,B 0,C 180,E1 -1338.962,E2 -1338.962} C_VEL
LIN {X 0,Y 587.34,Z 410.318,A -85,B 0,C 180,E1 -1341.744,E2 -1341.744} C_VEL
LIN {X 0,Y 587.349,Z 410.326,A -85,B 0,C 180,E1 -1344.507,E2 -1344.507} C_VEL
LIN {X 0,Y 587.351,Z 410.316,A -85,B 0,C 180,E1 -1347.256,E2 -1347.256} C_VEL
LIN {X 0,Y 587.384,Z 410.315,A -85,B 0,C 180,E1 -1350,E2 -1350} C_VEL
LIN {X 0,Y 587.365,Z 410.32,A -85,B 0,C 180,E1 -1352.743,E2 -1352.743} C_VEL
LIN {X 0,Y 587.338,Z 410.317,A -85,B 0,C 180,E1 -1355.493,E2 -1355.493} C_VEL
LIN {X 0,Y 587.315,Z 410.32,A -85,B 0,C 180,E1 -1357.564,E2 -1357.564} C_VEL
LIN {X 0,Y 587.335,Z 410.325,A -85,B 0,C 180,E1 -1360.34,E2 -1360.34} C_VEL
LIN {X 0,Y 587.306,Z 410.323,A -85,B 0,C 180,E1 -1363.142,E2 -1363.142} C_VEL
LIN {X 0,Y 587.321,Z 410.32,A -85,B 0,C 180,E1 -1365.263,E2 -1365.263} C_VEL
LIN {X 0,Y 587.311,Z 410.321,A -85,B 0,C 180,E1 -1367.407,E2 -1367.407} C_VEL
LIN {X 0,Y 587.309,Z 410.321,A -85,B 0,C 180,E1 -1369.576,E2 -1369.576} C_VEL
LIN {X 0,Y 587.316,Z 410.321,A -85,B 0,C 180,E1 -1371.774,E2 -1371.774} C_VEL
LIN {X 0,Y 587.346,Z 410.323,A -85,B 0,C 180,E1 -1374.759,E2 -1374.759} C_VEL
LIN {X 0,Y 587.3,Z 410.325,A -85,B 0,C 180,E1 -1377.047,E2 -1377.047} C_VEL
LIN {X 0,Y 587.341,Z 410.317,A -85,B 0,C 180,E1 -1379.38,E2 -1379.38} C_VEL
LIN {X 0,Y 587.342,Z 410.318,A -85,B 0,C 180,E1 -1381.835,E2 -1381.835} C_VEL
LIN {X 0,Y 587.341,Z 410.324,A -85,B 0,C 180,E1 -1384.346,E2 -1384.346} C_VEL
LIN {X 0,Y 587.341,Z 410.317,A -85,B 0,C 180,E1 -1387.608,E2 -1387.608} C_VEL
LIN {X 0,Y 587.31,Z 410.326,A -85,B 0,C 180,E1 -1390.254,E2 -1390.254} C_VEL
LIN {X 0,Y 587.302,Z 410.324,A -85,B 0,C 180,E1 -1393.117,E2 -1393.117} C_VEL
LIN {X 0,Y 587.312,Z 410.323,A -85,B 0,C 180,E1 -1396.048,E2 -1396.048} C_VEL
LIN {X 0,Y 587.332,Z 410.323,A -85,B 0,C 180,E1 -1398.925,E2 -1398.925} C_VEL
LIN {X 0,Y 587.318,Z 410.32,A -85,B 0,C 180,E1 -1401.52,E2 -1401.52} C_VEL
LIN {X 0,Y 587.288,Z 410.326,A -85,B 0,C 180,E1 -1404.1,E2 -1404.1} C_VEL
LIN {X 0,Y 587.334,Z 410.329,A -85,B 0,C 180,E1 -1406.603,E2 -1406.603} C_VEL
LIN {X 0,Y 587.334,Z 410.318,A -85,B 0,C 180,E1 -1409.491,E2 -1409.491} C_VEL
LIN {X 0,Y 587.34,Z 410.323,A -85,B 0,C 180,E1 -1412.309,E2 -1412.309} C_VEL
LIN {X 0,Y 587.353,Z 410.316,A -85,B 0,C 180,E1 -1415.42,E2 -1415.42} C_VEL
LIN {X 0,Y 587.316,Z 410.324,A -85,B 0,C 180,E1 -1418.225,E2 -1418.225} C_VEL
LIN {X 0,Y 587.34,Z 410.319,A -85,B 0,C 180,E1 -1421.151,E2 -1421.151} C_VEL
LIN {X 0,Y 587.32,Z 410.321,A -85,B 0,C 180,E1 -1423.31,E2 -1423.31} C_VEL
LIN {X 0,Y 587.359,Z 410.318,A -85,B 0,C 180,E1 -1426.154,E2 -1426.154} C_VEL
LIN {X 0,Y 587.337,Z 410.322,A -85,B 0,C 180,E1 -1428.962,E2 -1428.962} C_VEL
LIN {X 0,Y 587.362,Z 410.314,A -85,B 0,C 180,E1 -1431.745,E2 -1431.745} C_VEL
LIN {X 0,Y 587.363,Z 410.322,A -85,B 0,C 180,E1 -1434.507,E2 -1434.507} C_VEL
LIN {X 0,Y 587.358,Z 410.316,A -85,B 0,C 180,E1 -1437.257,E2 -1437.257} C_VEL
LIN {X 0,Y 587.383,Z 410.313,A -85,B 0,C 180,E1 -1440,E2 -1440} C_VEL
LIN {X 0,Y 587.374,Z 410.322,A -85,B 0,C 180,E1 -1442.743,E2 -1442.743} C_VEL
LIN {X 0,Y 587.344,Z 410.317,A -85,B 0,C 180,E1 -1445.493,E2 -1445.493} C_VEL
LIN {X 0,Y 587.366,Z 410.318,A -85,B 0,C 180,E1 -1448.255,E2 -1448.255} C_VEL
LIN {X 0,Y 587.349,Z 410.319,A -85,B 0,C 180,E1 -1451.134,E2 -1451.134} C_VEL
LIN {X 0,Y 587.366,Z 410.318,A -85,B 0,C 180,E1 -1454.26,E2 -1454.26} C_VEL
LIN {X 0,Y 587.347,Z 410.317,A -85,B 0,C 180,E1 -1457.406,E2 -1457.406} C_VEL
LIN {X 0,Y 587.328,Z 410.323,A -85,B 0,C 180,E1 -1460.305,E2 -1460.305} C_VEL
LIN {X 0,Y 587.315,Z 410.322,A -85,B 0,C 180,E1 -1463.259,E2 -1463.259} C_VEL
LIN {X 0,Y 587.322,Z 410.32,A -85,B 0,C 180,E1 -1465.517,E2 -1465.517} C_VEL
LIN {X 0,Y 587.306,Z 410.321,A -85,B 0,C 180,E1 -1467.82,E2 -1467.82} C_VEL
LIN {X 0,Y 587.336,Z 410.325,A -85,B 0,C 180,E1 -1470.51,E2 -1470.51} C_VEL
LIN {X 0,Y 587.328,Z 410.32,A -85,B 0,C 180,E1 -1473.397,E2 -1473.397} C_VEL
LIN {X 0,Y 587.298,Z 410.323,A -85,B 0,C 180,E1 -1475.9,E2 -1475.9} C_VEL
LIN {X 0,Y 587.329,Z 410.325,A -85,B 0,C 180,E1 -1478.48,E2 -1478.48} C_VEL
LIN {X 0,Y 587.333,Z 410.321,A -85,B 0,C 180,E1 -1481.157,E2 -1481.157} C_VEL
LIN {X 0,Y 587.327,Z 410.32,A -85,B 0,C 180,E1 -1484.114,E2 -1484.114} C_VEL
LIN {X 0,Y 587.319,Z 410.326,A -85,B 0,C 180,E1 -1486.994,E2 -1486.994} C_VEL
LIN {X 0,Y 587.316,Z 410.32,A -85,B 0,C 180,E1 -1489.746,E2 -1489.746} C_VEL
LIN {X 0,Y 587.345,Z 410.321,A -85,B 0,C 180,E1 -1492.393,E2 -1492.393} C_VEL
LIN {X 0,Y 587.358,Z 410.315,A -85,B 0,C 180,E1 -1495.78,E2 -1495.78} C_VEL
LIN {X 0,Y 587.339,Z 410.32,A -85,B 0,C 180,E1 -1498.231,E2 -1498.231} C_VEL
LIN {X 0,Y 587.346,Z 410.326,A -85,B 0,C 180,E1 -1500.868,E2 -1500.868} C_VEL
LIN {X 0,Y 587.331,Z 410.32,A -85,B 0,C 180,E1 -1503.721,E2 -1503.721} C_VEL
LIN {X 0,Y 587.333,Z 410.399,A -85,B 0,C 180,E1 -1505.273,E2 -1505.273} C_VEL
LIN {X 0,Y 588.057,Z 414.631,A -85,B 0,C 180,E1 -1505.86,E2 -1505.86} C_VEL
LIN {X 0,Y 587.846,Z 434.649,A -85,B 0,C 180,E1 -1508.443,E2 -1508.443} C_VEL
LIN {X 0,Y 587.72,Z 456.076,A -85,B 0,C 180,E1 -1511.164,E2 -1511.164} C_VEL
LIN {X 0,Y 587.569,Z 480.471,A -85,B 0,C 180,E1 -1514.21,E2 -1514.21} C_VEL
LIN {X 0,Y 587.398,Z 498.947,A -85,B 0,C 180,E1 -1516.486,E2 -1516.486} C_VEL
LIN {X 0,Y 587.841,Z 503.737,A -85,B 0,C 180,E1 -1516.563,E2 -1516.563} C_VEL
LIN {X 0,Y 587.716,Z 607.958,A -85,B 0,C 180,E1 -1517.855,E2 -1517.855} C_VEL
LIN {X 0,Y 587.676,Z 621.226,A -85,B 0,C 180,E1 -1518.161,E2 -1518.161} C_VEL
LIN {X 0,Y 587.593,Z 633.628,A -85,B 0,C 180,E1 -1518.585,E2 -1518.585} C_VEL
LIN {X 0,Y 587.55,Z 645.635,A -85,B 0,C 180,E1 -1519.141,E2 -1519.141} C_VEL
LIN {X 0,Y 587.453,Z 657.204,A -85,B 0,C 180,E1 -1519.837,E2 -1519.837} C_VEL
LIN {X 0,Y 587.393,Z 667.6,A -85,B 0,C 180,E1 -1520.618,E2 -1520.618} C_VEL
LIN {X 0,Y 587.321,Z 676.115,A -85,B 0,C 180,E1 -1521.398,E2 -1521.398} C_VEL
LIN {X 0,Y 587.274,Z 683.962,A -85,B 0,C 180,E1 -1522.263,E2 -1522.263} C_VEL
LIN {X 0,Y 587.23,Z 690.471,A -85,B 0,C 180,E1 -1523.127,E2 -1523.127} C_VEL
LIN {X 0,Y 587.236,Z 696.868,A -85,B 0,C 180,E1 -1524.162,E2 -1524.162} C_VEL
LIN {X 0,Y 587.147,Z 701.951,A -85,B 0,C 180,E1 -1525.194,E2 -1525.194} C_VEL
LIN {X 0,Y 587.213,Z 705.896,A -85,B 0,C 180,E1 -1526.226,E2 -1526.226} C_VEL
LIN {X 0,Y 587.132,Z 708.809,A -85,B 0,C 180,E1 -1527.256,E2 -1527.256} C_VEL
LIN {X 0,Y 587.14,Z 710.201,A -85,B 0,C 180,E1 -1527.942,E2 -1527.942} C_VEL
LIN {X 0,Y 587.14,Z 711.784,A -85,B 0,C 180,E1 -1529.314,E2 -1529.314} C_VEL
LIN {X 0,Y 587.137,Z 712,A -85,B 0,C 180,E1 -1530,E2 -1530} C_VEL
LIN {X 0,Y 587.147,Z 711.185,A -85,B 0,C 180,E1 -1531.372,E2 -1531.372} C_VEL
LIN {X 0,Y 587.14,Z 710.201,A -85,B 0,C 180,E1 -1532.058,E2 -1532.058} C_VEL
LIN {X 0,Y 587.132,Z 708.809,A -85,B 0,C 180,E1 -1532.745,E2 -1532.745} C_VEL
LIN {X 0,Y 587.213,Z 705.895,A -85,B 0,C 180,E1 -1533.775,E2 -1533.775} C_VEL
LIN {X 0,Y 587.147,Z 701.948,A -85,B 0,C 180,E1 -1534.807,E2 -1534.807} C_VEL
LIN {X 0,Y 587.217,Z 695.876,A -85,B 0,C 180,E1 -1536.011,E2 -1536.011} C_VEL
LIN {X 0,Y 587.245,Z 689.235,A -85,B 0,C 180,E1 -1537.046,E2 -1537.046} C_VEL
LIN {X 0,Y 587.3,Z 680.987,A -85,B 0,C 180,E1 -1538.083,E2 -1538.083} C_VEL
LIN {X 0,Y 587.343,Z 672.534,A -85,B 0,C 180,E1 -1538.949,E2 -1538.949} C_VEL
LIN {X 0,Y 587.419,Z 662.091,A -85,B 0,C 180,E1 -1539.817,E2 -1539.817} C_VEL
LIN {X 0,Y 587.508,Z 651.753,A -85,B 0,C 180,E1 -1540.511,E2 -1540.511} C_VEL
LIN {X 0,Y 587.568,Z 639.974,A -85,B 0,C 180,E1 -1541.141,E2 -1541.141} C_VEL
LIN {X 0,Y 587.61,Z 627.589,A -85,B 0,C 180,E1 -1541.64,E2 -1541.64} C_VEL
LIN {X 0,Y 587.691,Z 614.424,A -85,B 0,C 180,E1 -1542.015,E2 -1542.015} C_VEL
LIN {X 0,Y 587.743,Z 602.062,A -85,B 0,C 180,E1 -1542.232,E2 -1542.232} C_VEL
LIN {X 0,Y 587.724,Z 501.236,A -85,B 0,C 180,E1 -1543.471,E2 -1543.471} C_VEL
LIN {X 0,Y 587.4,Z 498.764,A -85,B 0,C 180,E1 -1543.536,E2 -1543.536} C_VEL
LIN {X 0,Y 587.585,Z 476.162,A -85,B 0,C 180,E1 -1546.325,E2 -1546.325} C_VEL
LIN {X 0,Y 587.73,Z 454.586,A -85,B 0,C 180,E1 -1549.024,E2 -1549.024} C_VEL
LIN {X 0,Y 587.869,Z 433.111,A -85,B 0,C 180,E1 -1551.753,E2 -1551.753} C_VEL
LIN {X 0,Y 588.058,Z 414.627,A -85,B 0,C 180,E1 -1554.141,E2 -1554.141} C_VEL
LIN {X 0,Y 587.311,Z 410.329,A -85,B 0,C 180,E1 -1554.761,E2 -1554.761} C_VEL
LIN {X 0,Y 587.332,Z 410.329,A -85,B 0,C 180,E1 -1557.046,E2 -1557.046} C_VEL
LIN {X 0,Y 587.349,Z 410.323,A -85,B 0,C 180,E1 -1559.38,E2 -1559.38} C_VEL
LIN {X 0,Y 587.345,Z 410.319,A -85,B 0,C 180,E1 -1561.835,E2 -1561.835} C_VEL
LIN {X 0,Y 587.352,Z 410.319,A -85,B 0,C 180,E1 -1564.348,E2 -1564.348} C_VEL
LIN {X 0,Y 587.348,Z 410.318,A -85,B 0,C 180,E1 -1567.608,E2 -1567.608} C_VEL
LIN {X 0,Y 587.315,Z 410.323,A -85,B 0,C 180,E1 -1570.255,E2 -1570.255} C_VEL
LIN {X 0,Y 587.308,Z 410.326,A -85,B 0,C 180,E1 -1573.117,E2 -1573.117} C_VEL
LIN {X 0,Y 587.317,Z 410.322,A -85,B 0,C 180,E1 -1576.049,E2 -1576.049} C_VEL
LIN {X 0,Y 587.336,Z 410.324,A -85,B 0,C 180,E1 -1578.926,E2 -1578.926} C_VEL
LIN {X 0,Y 587.321,Z 410.32,A -85,B 0,C 180,E1 -1581.52,E2 -1581.52} C_VEL
LIN {X 0,Y 587.284,Z 410.328,A -85,B 0,C 180,E1 -1584.099,E2 -1584.099} C_VEL
LIN {X 0,Y 587.336,Z 410.326,A -85,B 0,C 180,E1 -1586.603,E2 -1586.603} C_VEL
LIN {X 0,Y 587.321,Z 410.321,A -85,B 0,C 180,E1 -1589.033,E2 -1589.033} C_VEL
LIN {X 0,Y 587.309,Z 410.322,A -85,B 0,C 180,E1 -1591.402,E2 -1591.402} C_VEL
LIN {X 0,Y 587.312,Z 410.328,A -85,B 0,C 180,E1 -1594.482,E2 -1594.482} C_VEL
LIN {X 0,Y 587.307,Z 410.323,A -85,B 0,C 180,E1 -1597.485,E2 -1597.485} C_VEL
LIN {X 0,Y 587.287,Z 410.33,A -85,B 0,C 180,E1 -1600.423,E2 -1600.423} C_VEL
LIN {X 0,Y 587.292,Z 410.324,A -85,B 0,C 180,E1 -1603.309,E2 -1603.309} C_VEL
LIN {X 0,Y 587.338,Z 410.326,A -85,B 0,C 180,E1 -1606.154,E2 -1606.154} C_VEL
LIN {X 0,Y 587.255,Z 410.329,A -85,B 0,C 180,E1 -1608.961,E2 -1608.961} C_VEL
LIN {X 0,Y 587.327,Z 410.327,A -85,B 0,C 180,E1 -1611.744,E2 -1611.744} C_VEL
LIN {X 0,Y 587.324,Z 410.322,A -85,B 0,C 180,E1 -1614.507,E2 -1614.507} C_VEL
LIN {X 0,Y 587.344,Z 410.321,A -85,B 0,C 180,E1 -1617.257,E2 -1617.257} C_VEL
LIN {X 0,Y 587.36,Z 410.399,A -85,B 0,C 180,E1 -1619.143,E2 -1619.143} C_VEL
LIN {X 0,Y 587.285,Z 422.334,A -85,B 0,C 180,E1 -1621.564,E2 -1621.564} C_VEL
LIN {X 0,Y 587.857,Z 427.028,A -85,B 0,C 180,E1 -1621.648,E2 -1621.648} C_VEL
LIN {X 0,Y 587.698,Z 528.7,A -85,B 0,C 180,E1 -1622.913,E2 -1622.913} C_VEL
LIN {X 0,Y 587.654,Z 541.446,A -85,B 0,C 180,E1 -1623.214,E2 -1623.214} C_VEL
LIN {X 0,Y 587.593,Z 553.948,A -85,B 0,C 180,E1 -1623.643,E2 -1623.643} C_VEL
LIN {X 0,Y 587.522,Z 565.929,A -85,B 0,C 180,E1 -1624.202,E2 -1624.202} C_VEL
LIN {X 0,Y 587.402,Z 577.323,A -85,B 0,C 180,E1 -1624.89,E2 -1624.89} C_VEL
LIN {X 0,Y 587.4,Z 587.583,A -85,B 0,C 180,E1 -1625.665,E2 -1625.665} C_VEL
LIN {X 0,Y 587.339,Z 597.456,A -85,B 0,C 180,E1 -1626.58,E2 -1626.58} C_VEL
LIN {X 0,Y 587.263,Z 605.999,A -85,B 0,C 180,E1 -1627.564,E2 -1627.564} C_VEL
LIN {X 0,Y 587.248,Z 613.291,A -85,B 0,C 180,E1 -1628.603,E2 -1628.603} C_VEL
LIN {X 0,Y 587.2,Z 619.152,A -85,B 0,C 180,E1 -1629.646,E2 -1629.646} C_VEL
LIN {X 0,Y 587.189,Z 623.791,A -85,B 0,C 180,E1 -1630.691,E2 -1630.691} C_VEL
LIN {X 0,Y 587.163,Z 627.327,A -85,B 0,C 180,E1 -1631.741,E2 -1631.741} C_VEL
LIN {X 0,Y 587.158,Z 629.101,A -85,B 0,C 180,E1 -1632.442,E2 -1632.442} C_VEL
LIN {X 0,Y 587.146,Z 630.46,A -85,B 0,C 180,E1 -1633.146,E2 -1633.146} C_VEL
LIN {X 0,Y 587.144,Z 631.724,A -85,B 0,C 180,E1 -1634.288,E2 -1634.288} C_VEL
LIN {X 0,Y 587.126,Z 631.956,A -85,B 0,C 180,E1 -1635.269,E2 -1635.269} C_VEL
LIN {X 0,Y 587.138,Z 631.617,A -85,B 0,C 180,E1 -1635.98,E2 -1635.98} C_VEL
LIN {X 0,Y 587.148,Z 630.765,A -85,B 0,C 180,E1 -1636.747,E2 -1636.747} C_VEL
LIN {X 0,Y 587.129,Z 629.847,A -85,B 0,C 180,E1 -1637.271,E2 -1637.271} C_VEL
LIN {X 0,Y 586.468,Z 628.704,A -85,B 0,C 180,E1 -1637.833,E2 -1637.833} C_VEL
LIN {X 0,Y 583.607,Z 626.241,A -85,B 0,C 180,E1 -1638.731,E2 -1638.731} C_VEL
LIN {X 0,Y 581.196,Z 623.802,A -85,B 0,C 180,E1 -1639.439,E2 -1639.439} C_VEL
LIN {X 0,Y 580.176,Z 621.662,A -85,B 0,C 180,E1 -1639.976,E2 -1639.976} C_VEL
LIN {X 0,Y 580.102,Z 620.834,A -85,B 0,C 180,E1 -1640.156,E2 -1640.156} C_VEL
LIN {X 0,Y 580.153,Z 614.828,A -85,B 0,C 180,E1 -1641.31,E2 -1641.31} C_VEL
LIN {X 0,Y 580.186,Z 608.754,A -85,B 0,C 180,E1 -1642.243,E2 -1642.243} C_VEL
LIN {X 0,Y 580.235,Z 600.868,A -85,B 0,C 180,E1 -1643.237,E2 -1643.237} C_VEL
LIN {X 0,Y 580.314,Z 591.259,A -85,B 0,C 180,E1 -1644.221,E2 -1644.221} C_VEL
LIN {X 0,Y 580.415,Z 580.856,A -85,B 0,C 180,E1 -1645.075,E2 -1645.075} C_VEL
LIN {X 0,Y 580.472,Z 570.748,A -85,B 0,C 180,E1 -1645.744,E2 -1645.744} C_VEL
LIN {X 0,Y 580.607,Z 560.117,A -85,B 0,C 180,E1 -1646.311,E2 -1646.311} C_VEL
LIN {X 0,Y 580.686,Z 548.411,A -85,B 0,C 180,E1 -1646.797,E2 -1646.797} C_VEL
LIN {X 0,Y 580.762,Z 534.405,A -85,B 0,C 180,E1 -1647.207,E2 -1647.207} C_VEL
LIN {X 0,Y 580.821,Z 521.19,A -85,B 0,C 180,E1 -1647.437,E2 -1647.437} C_VEL
LIN {X 0,Y 580.793,Z 425.548,A -85,B 0,C 180,E1 -1648.626,E2 -1648.626} C_VEL
LIN {X 0,Y 580.247,Z 422.387,A -85,B 0,C 180,E1 -1648.682,E2 -1648.682} C_VEL
LIN {X 0,Y 580.286,Z 411.2,A -85,B 0,C 180,E1 -1651.01,E2 -1651.01} C_VEL
LIN {X 0,Y 580.308,Z 411.196,A -85,B 0,C 180,E1 -1653.855,E2 -1653.855} C_VEL
LIN {X 0,Y 580.274,Z 411.197,A -85,B 0,C 180,E1 -1657.27,E2 -1657.27} C_VEL
LIN {X 0,Y 580.287,Z 411.204,A -85,B 0,C 180,E1 -1660.269,E2 -1660.269} C_VEL
LIN {X 0,Y 580.273,Z 411.203,A -85,B 0,C 180,E1 -1662.707,E2 -1662.707} C_VEL
LIN {X 0,Y 580.253,Z 411.2,A -85,B 0,C 180,E1 -1665.611,E2 -1665.611} C_VEL
LIN {X 0,Y 580.251,Z 411.208,A -85,B 0,C 180,E1 -1668.228,E2 -1668.228} C_VEL
LIN {X 0,Y 580.268,Z 411.2,A -85,B 0,C 180,E1 -1670.964,E2 -1670.964} C_VEL
LIN {X 0,Y 580.242,Z 411.202,A -85,B 0,C 180,E1 -1673.594,E2 -1673.594} C_VEL
LIN {X 0,Y 580.312,Z 411.198,A -85,B 0,C 180,E1 -1676.145,E2 -1676.145} C_VEL
LIN {X 0,Y 580.269,Z 411.205,A -85,B 0,C 180,E1 -1678.614,E2 -1678.614} C_VEL
LIN {X 0,Y 580.285,Z 411.198,A -85,B 0,C 180,E1 -1681.023,E2 -1681.023} C_VEL
LIN {X 0,Y 580.266,Z 411.204,A -85,B 0,C 180,E1 -1684.149,E2 -1684.149} C_VEL
LIN {X 0,Y 580.259,Z 411.201,A -85,B 0,C 180,E1 -1686.999,E2 -1686.999} C_VEL
LIN {X 0,Y 580.266,Z 411.198,A -85,B 0,C 180,E1 -1689.437,E2 -1689.437} C_VEL
LIN {X 0,Y 580.247,Z 411.201,A -85,B 0,C 180,E1 -1691.644,E2 -1691.644} C_VEL
LIN {X 0,Y 580.277,Z 411.206,A -85,B 0,C 180,E1 -1694.546,E2 -1694.546} C_VEL
LIN {X 0,Y 580.251,Z 411.207,A -85,B 0,C 180,E1 -1696.695,E2 -1696.695} C_VEL
LIN {X 0,Y 580.308,Z 411.197,A -85,B 0,C 180,E1 -1698.827,E2 -1698.827} C_VEL
LIN {X 0,Y 580.307,Z 411.193,A -85,B 0,C 180,E1 -1701.643,E2 -1701.643} C_VEL
LIN {X 0,Y 580.315,Z 411.202,A -85,B 0,C 180,E1 -1704.44,E2 -1704.44} C_VEL
LIN {X 0,Y 580.32,Z 411.192,A -85,B 0,C 180,E1 -1707.223,E2 -1707.223} C_VEL
LIN {X 0,Y 580.353,Z 411.19,A -85,B 0,C 180,E1 -1710,E2 -1710} C_VEL
LIN {X 0,Y 580.329,Z 411.196,A -85,B 0,C 180,E1 -1712.776,E2 -1712.776} C_VEL
LIN {X 0,Y 580.307,Z 411.193,A -85,B 0,C 180,E1 -1715.56,E2 -1715.56} C_VEL
LIN {X 0,Y 580.269,Z 411.198,A -85,B 0,C 180,E1 -1717.656,E2 -1717.656} C_VEL
LIN {X 0,Y 580.295,Z 411.205,A -85,B 0,C 180,E1 -1720.467,E2 -1720.467} C_VEL
LIN {X 0,Y 580.264,Z 411.199,A -85,B 0,C 180,E1 -1723.304,E2 -1723.304} C_VEL
LIN {X 0,Y 580.286,Z 411.196,A -85,B 0,C 180,E1 -1725.453,E2 -1725.453} C_VEL
LIN {X 0,Y 580.27,Z 411.198,A -85,B 0,C 180,E1 -1727.625,E2 -1727.625} C_VEL
LIN {X 0,Y 580.285,Z 411.197,A -85,B 0,C 180,E1 -1729.823,E2 -1729.823} C_VEL
LIN {X 0,Y 580.268,Z 411.201,A -85,B 0,C 180,E1 -1732.053,E2 -1732.053} C_VEL
LIN {X 0,Y 580.299,Z 411.196,A -85,B 0,C 180,E1 -1735.08,E2 -1735.08} C_VEL
LIN {X 0,Y 580.281,Z 411.201,A -85,B 0,C 180,E1 -1738.186,E2 -1738.186} C_VEL
LIN {X 0,Y 580.281,Z 411.204,A -85,B 0,C 180,E1 -1740.694,E2 -1740.694} C_VEL
LIN {X 0,Y 580.283,Z 411.197,A -85,B 0,C 180,E1 -1743.313,E2 -1743.313} C_VEL
LIN {X 0,Y 580.243,Z 411.202,A -85,B 0,C 180,E1 -1745.756,E2 -1745.756} C_VEL
LIN {X 0,Y 580.287,Z 411.2,A -85,B 0,C 180,E1 -1748.146,E2 -1748.146} C_VEL
LIN {X 0,Y 580.294,Z 411.2,A -85,B 0,C 180,E1 -1750.844,E2 -1750.844} C_VEL
LIN {X 0,Y 580.241,Z 411.201,A -85,B 0,C 180,E1 -1753.661,E2 -1753.661} C_VEL
LIN {X 0,Y 580.266,Z 411.208,A -85,B 0,C 180,E1 -1756.61,E2 -1756.61} C_VEL
LIN {X 0,Y 580.295,Z 411.197,A -85,B 0,C 180,E1 -1759.156,E2 -1759.156} C_VEL
LIN {X 0,Y 580.286,Z 411.197,A -85,B 0,C 180,E1 -1761.927,E2 -1761.927} C_VEL
LIN {X 0,Y 580.248,Z 411.209,A -85,B 0,C 180,E1 -1764.452,E2 -1764.452} C_VEL
LIN {X 0,Y 580.288,Z 411.2,A -85,B 0,C 180,E1 -1766.975,E2 -1766.975} C_VEL
LIN {X 0,Y 580.293,Z 411.195,A -85,B 0,C 180,E1 -1769.425,E2 -1769.425} C_VEL
LIN {X 0,Y 580.288,Z 411.199,A -85,B 0,C 180,E1 -1772.143,E2 -1772.143} C_VEL
LIN {X 0,Y 580.321,Z 411.193,A -85,B 0,C 180,E1 -1775.27,E2 -1775.27} C_VEL
LIN {X 0,Y 580.266,Z 411.199,A -85,B 0,C 180,E1 -1777.947,E2 -1777.947} C_VEL
LIN {X 0,Y 580.291,Z 411.201,A -85,B 0,C 180,E1 -1780.913,E2 -1780.913} C_VEL
LIN {X 0,Y 580.262,Z 411.199,A -85,B 0,C 180,E1 -1783.825,E2 -1783.825} C_VEL
LIN {X 0,Y 580.268,Z 411.208,A -85,B 0,C 180,E1 -1786.696,E2 -1786.696} C_VEL
LIN {X 0,Y 580.306,Z 411.201,A -85,B 0,C 180,E1 -1788.827,E2 -1788.827} C_VEL
LIN {X 0,Y 580.325,Z 411.191,A -85,B 0,C 180,E1 -1791.644,E2 -1791.644} C_VEL
LIN {X 0,Y 580.329,Z 411.197,A -85,B 0,C 180,E1 -1794.44,E2 -1794.44} C_VEL
LIN {X 0,Y 580.326,Z 411.193,A -85,B 0,C 180,E1 -1797.223,E2 -1797.223} C_VEL
LIN {X 0,Y 580.352,Z 411.189,A -85,B 0,C 180,E1 -1800,E2 -1800} C_VEL
LIN {X 0,Y 580.339,Z 411.198,A -85,B 0,C 180,E1 -1802.777,E2 -1802.777} C_VEL
LIN {X 0,Y 580.312,Z 411.193,A -85,B 0,C 180,E1 -1805.56,E2 -1805.56} C_VEL
LIN {X 0,Y 580.317,Z 411.192,A -85,B 0,C 180,E1 -1807.656,E2 -1807.656} C_VEL
LIN {X 0,Y 580.301,Z 411.201,A -85,B 0,C 180,E1 -1810.467,E2 -1810.467} C_VEL
LIN {X 0,Y 580.27,Z 411.199,A -85,B 0,C 180,E1 -1813.304,E2 -1813.304} C_VEL
LIN {X 0,Y 580.29,Z 411.196,A -85,B 0,C 180,E1 -1815.453,E2 -1815.453} C_VEL
LIN {X 0,Y 580.292,Z 411.195,A -85,B 0,C 180,E1 -1817.625,E2 -1817.625} C_VEL
LIN {X 0,Y 580.287,Z 411.196,A -85,B 0,C 180,E1 -1819.823,E2 -1819.823} C_VEL
LIN {X 0,Y 580.27,Z 411.199,A -85,B 0,C 180,E1 -1822.053,E2 -1822.053} C_VEL
LIN {X 0,Y 580.301,Z 411.198,A -85,B 0,C 180,E1 -1825.08,E2 -1825.08} C_VEL
LIN {X 0,Y 580.282,Z 411.199,A -85,B 0,C 180,E1 -1828.187,E2 -1828.187} C_VEL
LIN {X 0,Y 580.284,Z 411.207,A -85,B 0,C 180,E1 -1830.695,E2 -1830.695} C_VEL
LIN {X 0,Y 580.283,Z 411.198,A -85,B 0,C 180,E1 -1833.313,E2 -1833.313} C_VEL
LIN {X 0,Y 580.251,Z 411.2,A -85,B 0,C 180,E1 -1835.757,E2 -1835.757} C_VEL
LIN {X 0,Y 580.288,Z 411.198,A -85,B 0,C 180,E1 -1838.147,E2 -1838.147} C_VEL
LIN {X 0,Y 580.297,Z 411.203,A -85,B 0,C 180,E1 -1840.844,E2 -1840.844} C_VEL
LIN {X 0,Y 580.279,Z 411.197,A -85,B 0,C 180,E1 -1843.658,E2 -1843.658} C_VEL
LIN {X 0,Y 580.282,Z 411.205,A -85,B 0,C 180,E1 -1846.609,E2 -1846.609} C_VEL
LIN {X 0,Y 580.299,Z 411.198,A -85,B 0,C 180,E1 -1849.157,E2 -1849.157} C_VEL
LIN {X 0,Y 580.289,Z 411.196,A -85,B 0,C 180,E1 -1851.928,E2 -1851.928} C_VEL
LIN {X 0,Y 580.251,Z 411.206,A -85,B 0,C 180,E1 -1854.453,E2 -1854.453} C_VEL
LIN {X 0,Y 580.29,Z 411.202,A -85,B 0,C 180,E1 -1856.975,E2 -1856.975} C_VEL
LIN {X 0,Y 580.296,Z 411.196,A -85,B 0,C 180,E1 -1859.425,E2 -1859.425} C_VEL
LIN {X 0,Y 580.297,Z 411.197,A -85,B 0,C 180,E1 -1862.142,E2 -1862.142} C_VEL
LIN {X 0,Y 580.293,Z 411.25,A -85,B 0,C 180,E1 -1865.066,E2 -1865.066} C_VEL
LIN {X 0,Y 581.218,Z 415.895,A -85,B 0,C 180,E1 -1865.725,E2 -1865.725} C_VEL
LIN {X 0,Y 580.967,Z 436.272,A -85,B 0,C 180,E1 -1868.386,E2 -1868.386} C_VEL
LIN {X 0,Y 580.794,Z 457.511,A -85,B 0,C 180,E1 -1871.114,E2 -1871.114} C_VEL
LIN {X 0,Y 580.588,Z 481.906,A -85,B 0,C 180,E1 -1874.195,E2 -1874.195} C_VEL
LIN {X 0,Y 580.43,Z 499.265,A -85,B 0,C 180,E1 -1876.332,E2 -1876.332} C_VEL
LIN {X 0,Y 580.931,Z 503.737,A -85,B 0,C 180,E1 -1876.4,E2 -1876.4} C_VEL
LIN {X 0,Y 580.797,Z 607.958,A -85,B 0,C 180,E1 -1877.708,E2 -1877.708} C_VEL
LIN {X 0,Y 580.735,Z 621.227,A -85,B 0,C 180,E1 -1878.017,E2 -1878.017} C_VEL
LIN {X 0,Y 580.644,Z 634.156,A -85,B 0,C 180,E1 -1878.467,E2 -1878.467} C_VEL
LIN {X 0,Y 580.556,Z 645.634,A -85,B 0,C 180,E1 -1879.009,E2 -1879.009} C_VEL
LIN {X 0,Y 580.428,Z 657.206,A -85,B 0,C 180,E1 -1879.712,E2 -1879.712} C_VEL
LIN {X 0,Y 580.344,Z 667.601,A -85,B 0,C 180,E1 -1880.503,E2 -1880.503} C_VEL
LIN {X 0,Y 580.271,Z 676.115,A -85,B 0,C 180,E1 -1881.292,E2 -1881.292} C_VEL
LIN {X 0,Y 580.222,Z 683.962,A -85,B 0,C 180,E1 -1882.168,E2 -1882.168} C_VEL
LIN {X 0,Y 580.153,Z 691.651,A -85,B 0,C 180,E1 -1883.222,E2 -1883.222} C_VEL
LIN {X 0,Y 580.139,Z 698.681,A -85,B 0,C 180,E1 -1884.439,E2 -1884.439} C_VEL
LIN {X 0,Y 580.108,Z 703.373,A -85,B 0,C 180,E1 -1885.484,E2 -1885.484} C_VEL
LIN {X 0,Y 580.123,Z 706.958,A -85,B 0,C 180,E1 -1886.528,E2 -1886.528} C_VEL
LIN {X 0,Y 580.043,Z 708.809,A -85,B 0,C 180,E1 -1887.222,E2 -1887.222} C_VEL
LIN {X 0,Y 580.039,Z 710.2,A -85,B 0,C 180,E1 -1887.917,E2 -1887.917} C_VEL
LIN {X 0,Y 580.04,Z 711.785,A -85,B 0,C 180,E1 -1889.306,E2 -1889.306} C_VEL
LIN {X 0,Y 580.037,Z 712,A -85,B 0,C 180,E1 -1890,E2 -1890} C_VEL
LIN {X 0,Y 580.046,Z 711.185,A -85,B 0,C 180,E1 -1891.389,E2 -1891.389} C_VEL
LIN {X 0,Y 580.039,Z 710.2,A -85,B 0,C 180,E1 -1892.083,E2 -1892.083} C_VEL
LIN {X 0,Y 580.043,Z 708.809,A -85,B 0,C 180,E1 -1892.778,E2 -1892.778} C_VEL
LIN {X 0,Y 580.11,Z 705.895,A -85,B 0,C 180,E1 -1893.821,E2 -1893.821} C_VEL
LIN {X 0,Y 580.053,Z 701.948,A -85,B 0,C 180,E1 -1894.866,E2 -1894.866} C_VEL
LIN {X 0,Y 580.139,Z 695.876,A -85,B 0,C 180,E1 -1896.085,E2 -1896.085} C_VEL
LIN {X 0,Y 580.184,Z 689.235,A -85,B 0,C 180,E1 -1897.133,E2 -1897.133} C_VEL
LIN {X 0,Y 580.251,Z 680.988,A -85,B 0,C 180,E1 -1898.182,E2 -1898.182} C_VEL
LIN {X 0,Y 580.308,Z 672.535,A -85,B 0,C 180,E1 -1899.059,E2 -1899.059} C_VEL
LIN {X 0,Y 580.419,Z 662.092,A -85,B 0,C 180,E1 -1899.936,E2 -1899.936} C_VEL
LIN {X 0,Y 580.513,Z 651.752,A -85,B 0,C 180,E1 -1900.64,E2 -1900.64} C_VEL
LIN {X 0,Y 580.581,Z 640.405,A -85,B 0,C 180,E1 -1901.256,E2 -1901.256} C_VEL
LIN {X 0,Y 580.65,Z 628.759,A -85,B 0,C 180,E1 -1901.741,E2 -1901.741} C_VEL
LIN {X 0,Y 580.749,Z 615.337,A -85,B 0,C 180,E1 -1902.138,E2 -1902.138} C_VEL
LIN {X 0,Y 580.817,Z 602.062,A -85,B 0,C 180,E1 -1902.381,E2 -1902.381} C_VEL
LIN {X 0,Y 580.86,Z 502.076,A -85,B 0,C 180,E1 -1903.623,E2 -1903.623} C_VEL
LIN {X 0,Y 580.408,Z 498.943,A -85,B 0,C 180,E1 -1903.68,E2 -1903.68} C_VEL
LIN {X 0,Y 580.626,Z 476.162,A -85,B 0,C 180,E1 -1906.526,E2 -1906.526} C_VEL
LIN {X 0,Y 580.8,Z 454.333,A -85,B 0,C 180,E1 -1909.292,E2 -1909.292} C_VEL
LIN {X 0,Y 581.026,Z 433.111,A -85,B 0,C 180,E1 -1912.023,E2 -1912.023} C_VEL
LIN {X 0,Y 581.209,Z 415.891,A -85,B 0,C 180,E1 -1914.276,E2 -1914.276} C_VEL
LIN {X 0,Y 580.263,Z 411.209,A -85,B 0,C 180,E1 -1914.976,E2 -1914.976} C_VEL
LIN {X 0,Y 580.3,Z 411.197,A -85,B 0,C 180,E1 -1917.858,E2 -1917.858} C_VEL
LIN {X 0,Y 580.288,Z 411.202,A -85,B 0,C 180,E1 -1920.695,E2 -1920.695} C_VEL
LIN {X 0,Y 580.305,Z 411.2,A -85,B 0,C 180,E1 -1923.316,E2 -1923.316} C_VEL
LIN {X 0,Y 580.25,Z 411.202,A -85,B 0,C 180,E1 -1925.756,E2 -1925.756} C_VEL
LIN {X 0,Y 580.292,Z 411.197,A -85,B 0,C 180,E1 -1928.146,E2 -1928.146} C_VEL
LIN {X 0,Y 580.3,Z 411.205,A -85,B 0,C 180,E1 -1930.844,E2 -1930.844} C_VEL
LIN {X 0,Y 580.273,Z 411.198,A -85,B 0,C 180,E1 -1933.659,E2 -1933.659} C_VEL
LIN {X 0,Y 580.272,Z 411.207,A -85,B 0,C 180,E1 -1936.61,E2 -1936.61} C_VEL
LIN {X 0,Y 580.299,Z 411.197,A -85,B 0,C 180,E1 -1939.156,E2 -1939.156} C_VEL
LIN {X 0,Y 580.29,Z 411.197,A -85,B 0,C 180,E1 -1941.928,E2 -1941.928} C_VEL
LIN {X 0,Y 580.236,Z 411.212,A -85,B 0,C 180,E1 -1944.451,E2 -1944.451} C_VEL
LIN {X 0,Y 580.29,Z 411.198,A -85,B 0,C 180,E1 -1946.975,E2 -1946.975} C_VEL
LIN {X 0,Y 580.284,Z 411.197,A -85,B 0,C 180,E1 -1949.424,E2 -1949.424} C_VEL
LIN {X 0,Y 580.256,Z 411.207,A -85,B 0,C 180,E1 -1952.15,E2 -1952.15} C_VEL
LIN {X 0,Y 580.278,Z 411.199,A -85,B 0,C 180,E1 -1954.919,E2 -1954.919} C_VEL
LIN {X 0,Y 580.249,Z 411.207,A -85,B 0,C 180,E1 -1957.946,E2 -1957.946} C_VEL
LIN {X 0,Y 580.227,Z 411.205,A -85,B 0,C 180,E1 -1960.871,E2 -1960.871} C_VEL
LIN {X 0,Y 580.231,Z 411.204,A -85,B 0,C 180,E1 -1963.114,E2 -1963.114} C_VEL
LIN {X 0,Y 580.3,Z 411.205,A -85,B 0,C 180,E1 -1965.982,E2 -1965.982} C_VEL
LIN {X 0,Y 580.25,Z 411.202,A -85,B 0,C 180,E1 -1968.837,E2 -1968.837} C_VEL
LIN {X 0,Y 580.294,Z 411.202,A -85,B 0,C 180,E1 -1971.643,E2 -1971.643} C_VEL
LIN {X 0,Y 580.293,Z 411.198,A -85,B 0,C 180,E1 -1974.44,E2 -1974.44} C_VEL
LIN {X 0,Y 580.311,Z 411.197,A -85,B 0,C 180,E1 -1977.223,E2 -1977.223} C_VEL
LIN {X 0,Y 580.313,Z 411.308,A -85,B 0,C 180,E1 -1979.133,E2 -1979.133} C_VEL
LIN {X 0,Y 580.243,Z 422.394,A -85,B 0,C 180,E1 -1981.41,E2 -1981.41} C_VEL
LIN {X 0,Y 580.969,Z 427.675,A -85,B 0,C 180,E1 -1981.495,E2 -1981.495} C_VEL
LIN {X 0,Y 580.788,Z 527.955,A -85,B 0,C 180,E1 -1982.753,E2 -1982.753} C_VEL
LIN {X 0,Y 580.696,Z 540.222,A -85,B 0,C 180,E1 -1983.035,E2 -1983.035} C_VEL
LIN {X 0,Y 580.656,Z 551.931,A -85,B 0,C 180,E1 -1983.426,E2 -1983.426} C_VEL
LIN {X 0,Y 580.558,Z 564.445,A -85,B 0,C 180,E1 -1983.991,E2 -1983.991} C_VEL
LIN {X 0,Y 580.415,Z 576.18,A -85,B 0,C 180,E1 -1984.688,E2 -1984.688} C_VEL
LIN {X 0,Y 580.355,Z 586.643,A -85,B 0,C 180,E1 -1985.472,E2 -1985.472} C_VEL
LIN {X 0,Y 580.286,Z 595.271,A -85,B 0,C 180,E1 -1986.258,E2 -1986.258} C_VEL
LIN {X 0,Y 580.228,Z 603.253,A -85,B 0,C 180,E1 -1987.132,E2 -1987.132} C_VEL
LIN {X 0,Y 580.176,Z 611.116,A -85,B 0,C 180,E1 -1988.183,E2 -1988.183} C_VEL
LIN {X 0,Y 580.129,Z 618.31,A -85,B 0,C 180,E1 -1989.413,E2 -1989.413} C_VEL
LIN {X 0,Y 580.101,Z 623.116,A -85,B 0,C 180,E1 -1990.47,E2 -1990.47} C_VEL
LIN {X 0,Y 580.073,Z 626.809,A -85,B 0,C 180,E1 -1991.532,E2 -1991.532} C_VEL
LIN {X 0,Y 580.049,Z 629.49,A -85,B 0,C 180,E1 -1992.597,E2 -1992.597} C_VEL
LIN {X 0,Y 580.061,Z 630.742,A -85,B 0,C 180,E1 -1993.309,E2 -1993.309} C_VEL
LIN {X 0,Y 580.053,Z 631.709,A -85,B 0,C 180,E1 -1994.234,E2 -1994.234} C_VEL
LIN {X 0,Y 580.022,Z 631.9,A -85,B 0,C 180,E1 -1995.46,E2 -1995.46} C_VEL
LIN {X 0,Y 580.034,Z 631.462,A -85,B 0,C 180,E1 -1996.181,E2 -1996.181} C_VEL
LIN {X 0,Y 580.031,Z 629.871,A -85,B 0,C 180,E1 -1997.272,E2 -1997.272} C_VEL
LIN {X 0,Y 580.057,Z 627.405,A -85,B 0,C 180,E1 -1998.362,E2 -1998.362} C_VEL
LIN {X 0,Y 580.077,Z 623.745,A -85,B 0,C 180,E1 -1999.462,E2 -1999.462} C_VEL
LIN {X 0,Y 580.102,Z 620.834,A -85,B 0,C 180,E1 -2000.156,E2 -2000.156} C_VEL
LIN {X 0,Y 579.462,Z 618.387,A -85,B 0,C 180,E1 -2000.684,E2 -2000.684} C_VEL
LIN {X 0,Y 576.63,Z 613.936,A -85,B 0,C 180,E1 -2001.517,E2 -2001.517} C_VEL
LIN {X 0,Y 573.78,Z 608.831,A -85,B 0,C 180,E1 -2002.319,E2 -2002.319} C_VEL
LIN {X 0,Y 573.121,Z 605.356,A -85,B 0,C 180,E1 -2002.795,E2 -2002.795} C_VEL
LIN {X 0,Y 573.228,Z 597.89,A -85,B 0,C 180,E1 -2003.674,E2 -2003.674} C_VEL
LIN {X 0,Y 573.328,Z 589.017,A -85,B 0,C 180,E1 -2004.535,E2 -2004.535} C_VEL
LIN {X 0,Y 573.386,Z 579.004,A -85,B 0,C 180,E1 -2005.33,E2 -2005.33} C_VEL
LIN {X 0,Y 573.498,Z 568.924,A -85,B 0,C 180,E1 -2005.983,E2 -2005.983} C_VEL
LIN {X 0,Y 573.641,Z 557.532,A -85,B 0,C 180,E1 -2006.572,E2 -2006.572} C_VEL
LIN {X 0,Y 573.766,Z 543.777,A -85,B 0,C 180,E1 -2007.098,E2 -2007.098} C_VEL
LIN {X 0,Y 573.839,Z 531.68,A -85,B 0,C 180,E1 -2007.414,E2 -2007.414} C_VEL
LIN {X 0,Y 573.907,Z 515.618,A -85,B 0,C 180,E1 -2007.658,E2 -2007.658} C_VEL
LIN {X 0,Y 573.981,Z 426.913,A -85,B 0,C 180,E1 -2008.773,E2 -2008.773} C_VEL
LIN {X 0,Y 573.193,Z 422.307,A -85,B 0,C 180,E1 -2008.869,E2 -2008.869} C_VEL
LIN {X 0,Y 573.267,Z 412.074,A -85,B 0,C 180,E1 -2011.042,E2 -2011.042} C_VEL
LIN {X 0,Y 573.245,Z 412.074,A -85,B 0,C 180,E1 -2013.52,E2 -2013.52} C_VEL
LIN {X 0,Y 573.189,Z 412.085,A -85,B 0,C 180,E1 -2016.053,E2 -2016.053} C_VEL
LIN {X 0,Y 573.234,Z 412.079,A -85,B 0,C 180,E1 -2018.702,E2 -2018.702} C_VEL
LIN {X 0,Y 573.209,Z 412.077,A -85,B 0,C 180,E1 -2021.459,E2 -2021.459} C_VEL
LIN {X 0,Y 573.22,Z 412.086,A -85,B 0,C 180,E1 -2024.335,E2 -2024.335} C_VEL
LIN {X 0,Y 573.219,Z 412.076,A -85,B 0,C 180,E1 -2027.361,E2 -2027.361} C_VEL
LIN {X 0,Y 573.236,Z 412.084,A -85,B 0,C 180,E1 -2030.392,E2 -2030.392} C_VEL
LIN {X 0,Y 573.223,Z 412.077,A -85,B 0,C 180,E1 -2033.075,E2 -2033.075} C_VEL
LIN {X 0,Y 573.262,Z 412.072,A -85,B 0,C 180,E1 -2035.671,E2 -2035.671} C_VEL
LIN {X 0,Y 573.238,Z 412.08,A -85,B 0,C 180,E1 -2038.184,E2 -2038.184} C_VEL
LIN {X 0,Y 573.243,Z 412.08,A -85,B 0,C 180,E1 -2040.633,E2 -2040.633} C_VEL
LIN {X 0,Y 573.211,Z 412.077,A -85,B 0,C 180,E1 -2043.513,E2 -2043.513} C_VEL
LIN {X 0,Y 573.216,Z 412.082,A -85,B 0,C 180,E1 -2046.134,E2 -2046.134} C_VEL
LIN {X 0,Y 573.248,Z 412.073,A -85,B 0,C 180,E1 -2049.173,E2 -2049.173} C_VEL
LIN {X 0,Y 573.204,Z 412.078,A -85,B 0,C 180,E1 -2051.41,E2 -2051.41} C_VEL
LIN {X 0,Y 573.221,Z 412.076,A -85,B 0,C 180,E1 -2053.621,E2 -2053.621} C_VEL
LIN {X 0,Y 573.26,Z 412.072,A -85,B 0,C 180,E1 -2055.806,E2 -2055.806} C_VEL
LIN {X 0,Y 573.266,Z 412.076,A -85,B 0,C 180,E1 -2058.745,E2 -2058.745} C_VEL
LIN {X 0,Y 573.251,Z 412.072,A -85,B 0,C 180,E1 -2061.54,E2 -2061.54} C_VEL
LIN {X 0,Y 573.283,Z 412.077,A -85,B 0,C 180,E1 -2064.371,E2 -2064.371} C_VEL
LIN {X 0,Y 573.311,Z 412.067,A -85,B 0,C 180,E1 -2067.892,E2 -2067.892} C_VEL
LIN {X 0,Y 573.328,Z 412.069,A -85,B 0,C 180,E1 -2070.702,E2 -2070.702} C_VEL
LIN {X 0,Y 573.295,Z 412.072,A -85,B 0,C 180,E1 -2072.81,E2 -2072.81} C_VEL
LIN {X 0,Y 573.276,Z 412.069,A -85,B 0,C 180,E1 -2075.628,E2 -2075.628} C_VEL
LIN {X 0,Y 573.225,Z 412.076,A -85,B 0,C 180,E1 -2077.751,E2 -2077.751} C_VEL
LIN {X 0,Y 573.263,Z 412.08,A -85,B 0,C 180,E1 -2080.596,E2 -2080.596} C_VEL
LIN {X 0,Y 573.239,Z 412.08,A -85,B 0,C 180,E1 -2082.749,E2 -2082.749} C_VEL
LIN {X 0,Y 573.232,Z 412.078,A -85,B 0,C 180,E1 -2084.92,E2 -2084.92} C_VEL
LIN {X 0,Y 573.23,Z 412.076,A -85,B 0,C 180,E1 -2087.849,E2 -2087.849} C_VEL
LIN {X 0,Y 573.241,Z 412.077,A -85,B 0,C 180,E1 -2090.077,E2 -2090.077} C_VEL
LIN {X 0,Y 573.232,Z 412.082,A -85,B 0,C 180,E1 -2092.338,E2 -2092.338} C_VEL
LIN {X 0,Y 573.243,Z 412.073,A -85,B 0,C 180,E1 -2095.41,E2 -2095.41} C_VEL
LIN {X 0,Y 573.227,Z 412.085,A -85,B 0,C 180,E1 -2098.565,E2 -2098.565} C_VEL
LIN {X 0,Y 573.223,Z 412.079,A -85,B 0,C 180,E1 -2100.993,E2 -2100.993} C_VEL
LIN {X 0,Y 573.263,Z 412.071,A -85,B 0,C 180,E1 -2103.524,E2 -2103.524} C_VEL
LIN {X 0,Y 573.193,Z 412.082,A -85,B 0,C 180,E1 -2106.053,E2 -2106.053} C_VEL
LIN {X 0,Y 573.238,Z 412.082,A -85,B 0,C 180,E1 -2108.702,E2 -2108.702} C_VEL
LIN {X 0,Y 573.227,Z 412.075,A -85,B 0,C 180,E1 -2111.592,E2 -2111.592} C_VEL
LIN {X 0,Y 573.215,Z 412.085,A -85,B 0,C 180,E1 -2114.674,E2 -2114.674} C_VEL
LIN {X 0,Y 573.235,Z 412.074,A -85,B 0,C 180,E1 -2117.599,E2 -2117.599} C_VEL
LIN {X 0,Y 573.24,Z 412.084,A -85,B 0,C 180,E1 -2120.569,E2 -2120.569} C_VEL
LIN {X 0,Y 573.23,Z 412.078,A -85,B 0,C 180,E1 -2123.076,E2 -2123.076} C_VEL
LIN {X 0,Y 573.263,Z 412.071,A -85,B 0,C 180,E1 -2125.671,E2 -2125.671} C_VEL
LIN {X 0,Y 573.237,Z 412.078,A -85,B 0,C 180,E1 -2128.184,E2 -2128.184} C_VEL
LIN {X 0,Y 573.26,Z 412.081,A -85,B 0,C 180,E1 -2130.634,E2 -2130.634} C_VEL
LIN {X 0,Y 573.209,Z 412.081,A -85,B 0,C 180,E1 -2133.022,E2 -2133.022} C_VEL
LIN {X 0,Y 573.275,Z 412.07,A -85,B 0,C 180,E1 -2135.366,E2 -2135.366} C_VEL
LIN {X 0,Y 573.227,Z 412.082,A -85,B 0,C 180,E1 -2138.419,E2 -2138.419} C_VEL
LIN {X 0,Y 573.269,Z 412.078,A -85,B 0,C 180,E1 -2140.731,E2 -2140.731} C_VEL
LIN {X 0,Y 573.238,Z 412.074,A -85,B 0,C 180,E1 -2143.621,E2 -2143.621} C_VEL
LIN {X 0,Y 573.259,Z 412.072,A -85,B 0,C 180,E1 -2145.807,E2 -2145.807} C_VEL
LIN {X 0,Y 573.263,Z 412.079,A -85,B 0,C 180,E1 -2148.745,E2 -2148.745} C_VEL
LIN {X 0,Y 573.281,Z 412.069,A -85,B 0,C 180,E1 -2151.54,E2 -2151.54} C_VEL
LIN {X 0,Y 573.295,Z 412.072,A -85,B 0,C 180,E1 -2154.372,E2 -2154.372} C_VEL
LIN {X 0,Y 573.311,Z 412.065,A -85,B 0,C 180,E1 -2157.892,E2 -2157.892} C_VEL
LIN {X 0,Y 573.333,Z 412.072,A -85,B 0,C 180,E1 -2160.702,E2 -2160.702} C_VEL
LIN {X 0,Y 573.304,Z 412.073,A -85,B 0,C 180,E1 -2162.811,E2 -2162.811} C_VEL
LIN {X 0,Y 573.281,Z 412.068,A -85,B 0,C 180,E1 -2165.628,E2 -2165.628} C_VEL
LIN {X 0,Y 573.269,Z 412.07,A -85,B 0,C 180,E1 -2167.75,E2 -2167.75} C_VEL
LIN {X 0,Y 573.267,Z 412.079,A -85,B 0,C 180,E1 -2170.597,E2 -2170.597} C_VEL
LIN {X 0,Y 573.263,Z 412.08,A -85,B 0,C 180,E1 -2172.749,E2 -2172.749} C_VEL
LIN {X 0,Y 573.233,Z 412.081,A -85,B 0,C 180,E1 -2174.92,E2 -2174.92} C_VEL
LIN {X 0,Y 573.243,Z 412.073,A -85,B 0,C 180,E1 -2177.849,E2 -2177.849} C_VEL
LIN {X 0,Y 573.242,Z 412.075,A -85,B 0,C 180,E1 -2180.077,E2 -2180.077} C_VEL
LIN {X 0,Y 573.233,Z 412.079,A -85,B 0,C 180,E1 -2182.338,E2 -2182.338} C_VEL
LIN {X 0,Y 573.245,Z 412.074,A -85,B 0,C 180,E1 -2185.411,E2 -2185.411} C_VEL
LIN {X 0,Y 573.229,Z 412.083,A -85,B 0,C 180,E1 -2188.565,E2 -2188.565} C_VEL
LIN {X 0,Y 573.225,Z 412.081,A -85,B 0,C 180,E1 -2190.994,E2 -2190.994} C_VEL
LIN {X 0,Y 573.263,Z 412.071,A -85,B 0,C 180,E1 -2193.524,E2 -2193.524} C_VEL
LIN {X 0,Y 573.217,Z 412.078,A -85,B 0,C 180,E1 -2196.052,E2 -2196.052} C_VEL
LIN {X 0,Y 573.241,Z 412.084,A -85,B 0,C 180,E1 -2198.702,E2 -2198.702} C_VEL
LIN {X 0,Y 573.23,Z 412.075,A -85,B 0,C 180,E1 -2201.593,E2 -2201.593} C_VEL
LIN {X 0,Y 573.234,Z 412.078,A -85,B 0,C 180,E1 -2204.334,E2 -2204.334} C_VEL
LIN {X 0,Y 573.243,Z 412.075,A -85,B 0,C 180,E1 -2207.359,E2 -2207.359} C_VEL
LIN {X 0,Y 573.25,Z 412.08,A -85,B 0,C 180,E1 -2210.568,E2 -2210.568} C_VEL
LIN {X 0,Y 573.233,Z 412.079,A -85,B 0,C 180,E1 -2213.076,E2 -2213.076} C_VEL
LIN {X 0,Y 573.266,Z 412.07,A -85,B 0,C 180,E1 -2215.671,E2 -2215.671} C_VEL
LIN {X 0,Y 573.24,Z 412.076,A -85,B 0,C 180,E1 -2218.185,E2 -2218.185} C_VEL
LIN {X 0,Y 573.262,Z 412.08,A -85,B 0,C 180,E1 -2220.634,E2 -2220.634} C_VEL
LIN {X 0,Y 573.249,Z 412.081,A -85,B 0,C 180,E1 -2223.024,E2 -2223.024} C_VEL
LIN {X 0,Y 573.258,Z 412.086,A -85,B 0,C 180,E1 -2224.889,E2 -2224.889} C_VEL
LIN {X 0,Y 574.329,Z 417.275,A -85,B 0,C 180,E1 -2225.607,E2 -2225.607} C_VEL
LIN {X 0,Y 574.08,Z 435.985,A -85,B 0,C 180,E1 -2228.076,E2 -2228.076} C_VEL
LIN {X 0,Y 573.88,Z 455.047,A -85,B 0,C 180,E1 -2230.558,E2 -2230.558} C_VEL
LIN {X 0,Y 573.641,Z 477.603,A -85,B 0,C 180,E1 -2233.451,E2 -2233.451} C_VEL
LIN {X 0,Y 573.428,Z 498.947,A -85,B 0,C 180,E1 -2236.15,E2 -2236.15} C_VEL
LIN {X 0,Y 574.05,Z 505.526,A -85,B 0,C 180,E1 -2236.256,E2 -2236.256} C_VEL
LIN {X 0,Y 573.881,Z 607.958,A -85,B 0,C 180,E1 -2237.558,E2 -2237.558} C_VEL
LIN {X 0,Y 573.794,Z 621.227,A -85,B 0,C 180,E1 -2237.87,E2 -2237.87} C_VEL
LIN {X 0,Y 573.691,Z 634.157,A -85,B 0,C 180,E1 -2238.325,E2 -2238.325} C_VEL
LIN {X 0,Y 573.591,Z 645.634,A -85,B 0,C 180,E1 -2238.874,E2 -2238.874} C_VEL
LIN {X 0,Y 573.44,Z 657.206,A -85,B 0,C 180,E1 -2239.585,E2 -2239.585} C_VEL
LIN {X 0,Y 573.331,Z 667.603,A -85,B 0,C 180,E1 -2240.386,E2 -2240.386} C_VEL
LIN {X 0,Y 573.241,Z 676.115,A -85,B 0,C 180,E1 -2241.185,E2 -2241.185} C_VEL
LIN {X 0,Y 573.161,Z 683.962,A -85,B 0,C 180,E1 -2242.071,E2 -2242.071} C_VEL
LIN {X 0,Y 573.072,Z 691.955,A -85,B 0,C 180,E1 -2243.186,E2 -2243.186} C_VEL
LIN {X 0,Y 573.07,Z 698.681,A -85,B 0,C 180,E1 -2244.37,E2 -2244.37} C_VEL
LIN {X 0,Y 573.028,Z 703.373,A -85,B 0,C 180,E1 -2245.428,E2 -2245.428} C_VEL
LIN {X 0,Y 573.022,Z 706.958,A -85,B 0,C 180,E1 -2246.484,E2 -2246.484} C_VEL
LIN {X 0,Y 572.959,Z 708.809,A -85,B 0,C 180,E1 -2247.188,E2 -2247.188} C_VEL
LIN {X 0,Y 572.939,Z 710.199,A -85,B 0,C 180,E1 -2247.891,E2 -2247.891} C_VEL
LIN {X 0,Y 572.94,Z 711.785,A -85,B 0,C 180,E1 -2249.297,E2 -2249.297} C_VEL
LIN {X 0,Y 572.938,Z 712,A -85,B 0,C 180,E1 -2250,E2 -2250} C_VEL
LIN {X 0,Y 572.946,Z 711.186,A -85,B 0,C 180,E1 -2251.406,E2 -2251.406} C_VEL
LIN {X 0,Y 572.939,Z 710.199,A -85,B 0,C 180,E1 -2252.109,E2 -2252.109} C_VEL
LIN {X 0,Y 572.959,Z 708.809,A -85,B 0,C 180,E1 -2252.813,E2 -2252.813} C_VEL
LIN {X 0,Y 573.015,Z 705.895,A -85,B 0,C 180,E1 -2253.868,E2 -2253.868} C_VEL
LIN {X 0,Y 572.963,Z 701.948,A -85,B 0,C 180,E1 -2254.926,E2 -2254.926} C_VEL
LIN {X 0,Y 573.065,Z 695.875,A -85,B 0,C 180,E1 -2256.16,E2 -2256.16} C_VEL
LIN {X 0,Y 573.12,Z 689.236,A -85,B 0,C 180,E1 -2257.221,E2 -2257.221} C_VEL
LIN {X 0,Y 573.201,Z 680.988,A -85,B 0,C 180,E1 -2258.283,E2 -2258.283} C_VEL
LIN {X 0,Y 573.287,Z 672.535,A -85,B 0,C 180,E1 -2259.171,E2 -2259.171} C_VEL
LIN {X 0,Y 573.424,Z 662.094,A -85,B 0,C 180,E1 -2260.059,E2 -2260.059} C_VEL
LIN {X 0,Y 573.556,Z 650.398,A -85,B 0,C 180,E1 -2260.855,E2 -2260.855} C_VEL
LIN {X 0,Y 573.653,Z 639.28,A -85,B 0,C 180,E1 -2261.447,E2 -2261.447} C_VEL
LIN {X 0,Y 573.724,Z 626.164,A -85,B 0,C 180,E1 -2261.975,E2 -2261.975} C_VEL
LIN {X 0,Y 573.836,Z 613.507,A -85,B 0,C 180,E1 -2262.332,E2 -2262.332} C_VEL
LIN {X 0,Y 573.897,Z 600.285,A -85,B 0,C 180,E1 -2262.555,E2 -2262.555} C_VEL
LIN {X 0,Y 573.99,Z 503.026,A -85,B 0,C 180,E1 -2263.777,E2 -2263.777} C_VEL
LIN {X 0,Y 573.416,Z 498.943,A -85,B 0,C 180,E1 -2263.85,E2 -2263.85} C_VEL
LIN {X 0,Y 573.665,Z 476.17,A -85,B 0,C 180,E1 -2266.732,E2 -2266.732} C_VEL
LIN {X 0,Y 573.863,Z 455.088,A -85,B 0,C 180,E1 -2269.437,E2 -2269.437} C_VEL
LIN {X 0,Y 574.06,Z 437.416,A -85,B 0,C 180,E1 -2271.737,E2 -2271.737} C_VEL
LIN {X 0,Y 574.352,Z 418.748,A -85,B 0,C 180,E1 -2274.2,E2 -2274.2} C_VEL
LIN {X 0,Y 573.728,Z 414.325,A -85,B 0,C 180,E1 -2274.792,E2 -2274.792} C_VEL
LIN {X 0,Y 573.26,Z 412.082,A -85,B 0,C 180,E1 -2275.111,E2 -2275.111} C_VEL
LIN {X 0,Y 573.253,Z 412.074,A -85,B 0,C 180,E1 -2278.029,E2 -2278.029} C_VEL
LIN {X 0,Y 573.25,Z 412.075,A -85,B 0,C 180,E1 -2280.176,E2 -2280.176} C_VEL
LIN {X 0,Y 573.256,Z 412.078,A -85,B 0,C 180,E1 -2282.645,E2 -2282.645} C_VEL
LIN {X 0,Y 573.211,Z 412.085,A -85,B 0,C 180,E1 -2285.188,E2 -2285.188} C_VEL
LIN {X 0,Y 573.239,Z 412.075,A -85,B 0,C 180,E1 -2287.808,E2 -2287.808} C_VEL
LIN {X 0,Y 573.249,Z 412.079,A -85,B 0,C 180,E1 -2290.525,E2 -2290.525} C_VEL
LIN {X 0,Y 573.235,Z 412.077,A -85,B 0,C 180,E1 -2293.36,E2 -2293.36} C_VEL
LIN {X 0,Y 573.24,Z 412.078,A -85,B 0,C 180,E1 -2296.332,E2 -2296.332} C_VEL
LIN {X 0,Y 573.23,Z 412.084,A -85,B 0,C 180,E1 -2298.543,E2 -2298.543} C_VEL
LIN {X 0,Y 573.24,Z 412.075,A -85,B 0,C 180,E1 -2301.298,E2 -2301.298} C_VEL
LIN {X 0,Y 573.192,Z 412.083,A -85,B 0,C 180,E1 -2304.022,E2 -2304.022} C_VEL
LIN {X 0,Y 573.258,Z 412.081,A -85,B 0,C 180,E1 -2306.517,E2 -2306.517} C_VEL
LIN {X 0,Y 573.223,Z 412.077,A -85,B 0,C 180,E1 -2309.12,E2 -2309.12} C_VEL
